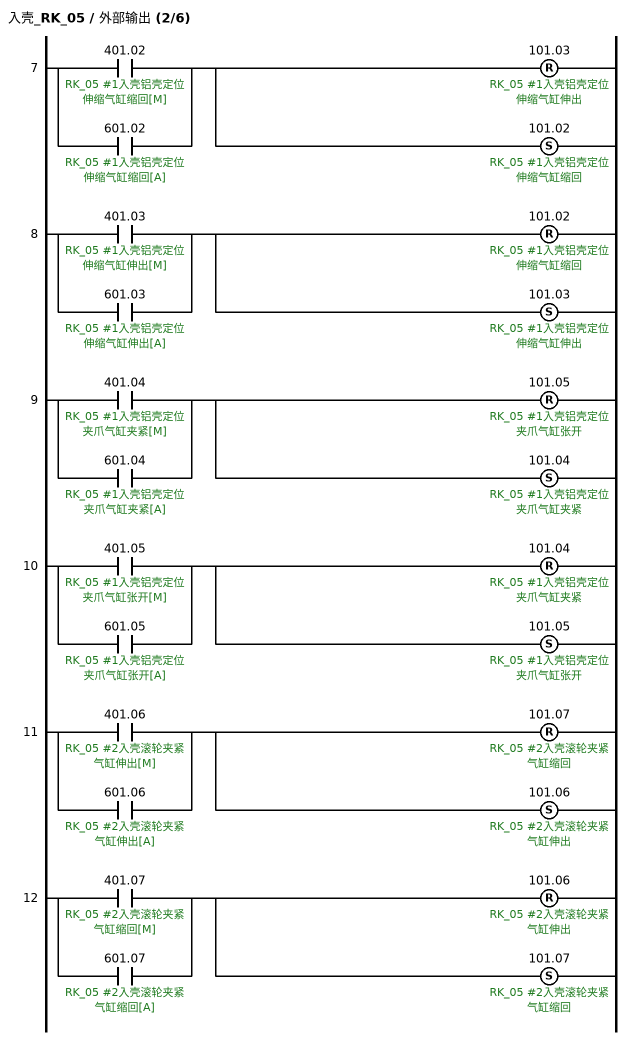
; [picture p504: 入壳_RK_05 / 外部输出, rungs 7-12]
; rung 7
LD 401.02  ; RK_05 #1入壳铝壳定位伸缩气缸缩回[M]
OR 601.02  ; RK_05 #1入壳铝壳定位伸缩气缸缩回[A]
RSET 101.03  ; RK_05 #1入壳铝壳定位伸缩气缸伸出
SET 101.02  ; RK_05 #1入壳铝壳定位伸缩气缸缩回
; rung 8
LD 401.03  ; RK_05 #1入壳铝壳定位伸缩气缸伸出[M]
OR 601.03  ; RK_05 #1入壳铝壳定位伸缩气缸伸出[A]
RSET 101.02  ; RK_05 #1入壳铝壳定位伸缩气缸缩回
SET 101.03  ; RK_05 #1入壳铝壳定位伸缩气缸伸出
; rung 9
LD 401.04  ; RK_05 #1入壳铝壳定位夹爪气缸夹紧[M]
OR 601.04  ; RK_05 #1入壳铝壳定位夹爪气缸夹紧[A]
RSET 101.05  ; RK_05 #1入壳铝壳定位夹爪气缸张开
SET 101.04  ; RK_05 #1入壳铝壳定位夹爪气缸夹紧
; rung 10
LD 401.05  ; RK_05 #1入壳铝壳定位夹爪气缸张开[M]
OR 601.05  ; RK_05 #1入壳铝壳定位夹爪气缸张开[A]
RSET 101.04  ; RK_05 #1入壳铝壳定位夹爪气缸夹紧
SET 101.05  ; RK_05 #1入壳铝壳定位夹爪气缸张开
; rung 11
LD 401.06  ; RK_05 #2入壳滚轮夹紧气缸伸出[M]
OR 601.06  ; RK_05 #2入壳滚轮夹紧气缸伸出[A]
RSET 101.07  ; RK_05 #2入壳滚轮夹紧气缸缩回
SET 101.06  ; RK_05 #2入壳滚轮夹紧气缸伸出
; rung 12
LD 401.07  ; RK_05 #2入壳滚轮夹紧气缸缩回[M]
OR 601.07  ; RK_05 #2入壳滚轮夹紧气缸缩回[A]
RSET 101.06  ; RK_05 #2入壳滚轮夹紧气缸伸出
SET 101.07  ; RK_05 #2入壳滚轮夹紧气缸缩回

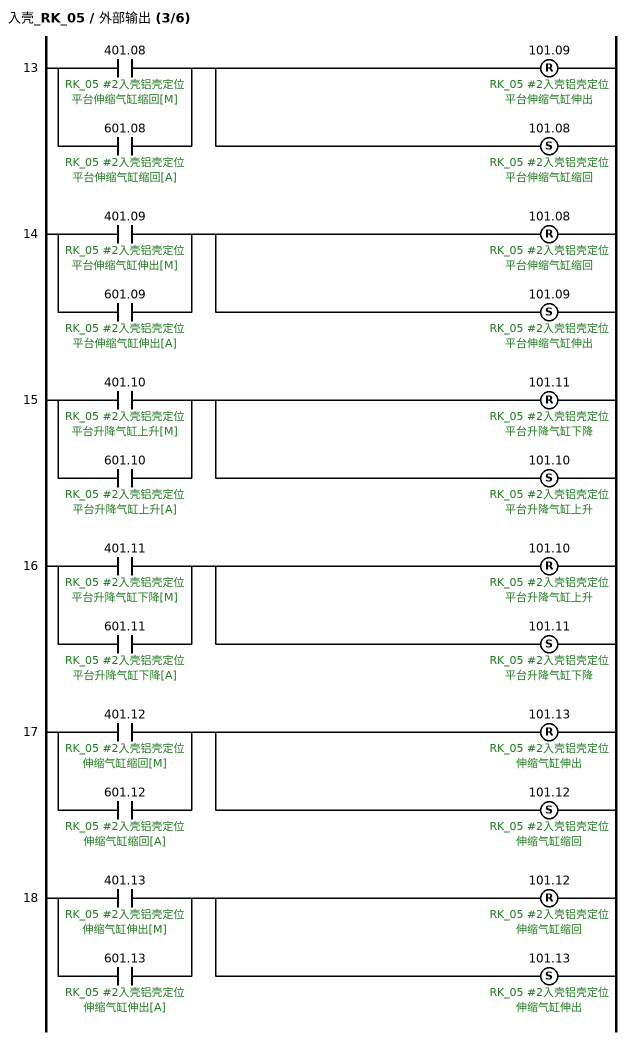
; rung 13
LD 401.08  ; RK_05 #2入壳铝壳定位平台伸缩气缸缩回[M]
OR 601.08  ; RK_05 #2入壳铝壳定位平台伸缩气缸缩回[A]
RSET 101.09  ; RK_05 #2入壳铝壳定位平台伸缩气缸伸出
SET 101.08  ; RK_05 #2入壳铝壳定位平台伸缩气缸缩回
; rung 14
LD 401.09  ; RK_05 #2入壳铝壳定位平台伸缩气缸伸出[M]
OR 601.09  ; RK_05 #2入壳铝壳定位平台伸缩气缸伸出[A]
RSET 101.08  ; RK_05 #2入壳铝壳定位平台伸缩气缸缩回
SET 101.09  ; RK_05 #2入壳铝壳定位平台伸缩气缸伸出
; rung 15
LD 401.10  ; RK_05 #2入壳铝壳定位平台升降气缸上升[M]
OR 601.10  ; RK_05 #2入壳铝壳定位平台升降气缸上升[A]
RSET 101.11  ; RK_05 #2入壳铝壳定位平台升降气缸下降
SET 101.10  ; RK_05 #2入壳铝壳定位平台升降气缸上升
; rung 16
LD 401.11  ; RK_05 #2入壳铝壳定位平台升降气缸下降[M]
OR 601.11  ; RK_05 #2入壳铝壳定位平台升降气缸下降[A]
RSET 101.10  ; RK_05 #2入壳铝壳定位平台升降气缸上升
SET 101.11  ; RK_05 #2入壳铝壳定位平台升降气缸下降
; rung 17
LD 401.12  ; RK_05 #2入壳铝壳定位伸缩气缸缩回[M]
OR 601.12  ; RK_05 #2入壳铝壳定位伸缩气缸缩回[A]
RSET 101.13  ; RK_05 #2入壳铝壳定位伸缩气缸伸出
SET 101.12  ; RK_05 #2入壳铝壳定位伸缩气缸缩回
; rung 18
LD 401.13  ; RK_05 #2入壳铝壳定位伸缩气缸伸出[M]
OR 601.13  ; RK_05 #2入壳铝壳定位伸缩气缸伸出[A]
RSET 101.12  ; RK_05 #2入壳铝壳定位伸缩气缸缩回
SET 101.13  ; RK_05 #2入壳铝壳定位伸缩气缸伸出

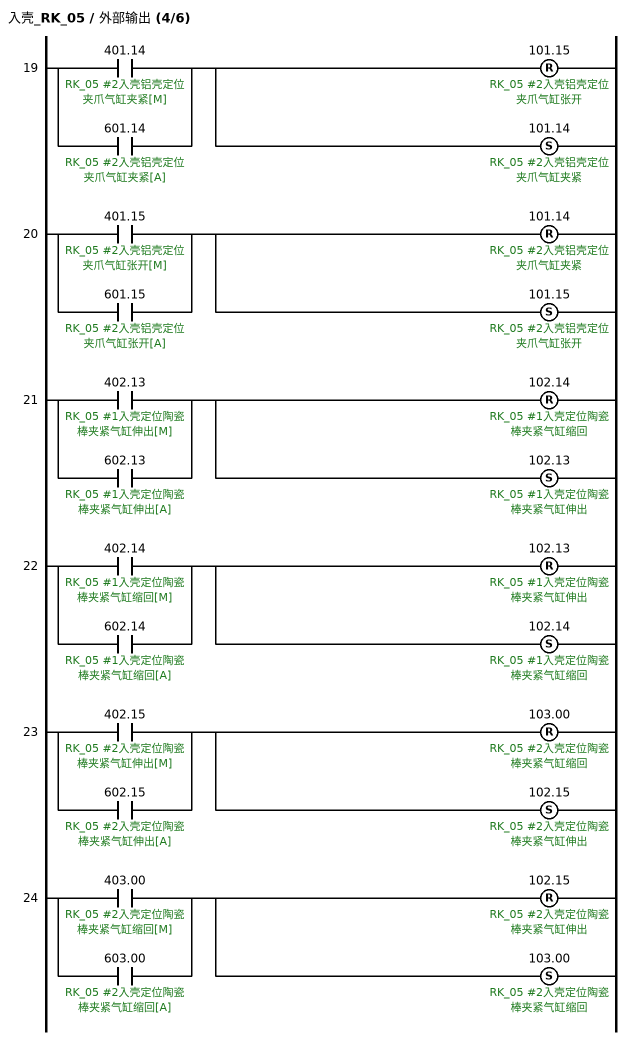
; rung 19
LD 401.14  ; RK_05 #2入壳铝壳定位夹爪气缸夹紧[M]
OR 601.14  ; RK_05 #2入壳铝壳定位夹爪气缸夹紧[A]
RSET 101.15  ; RK_05 #2入壳铝壳定位夹爪气缸张开
SET 101.14  ; RK_05 #2入壳铝壳定位夹爪气缸夹紧
; rung 20
LD 401.15  ; RK_05 #2入壳铝壳定位夹爪气缸张开[M]
OR 601.15  ; RK_05 #2入壳铝壳定位夹爪气缸张开[A]
RSET 101.14  ; RK_05 #2入壳铝壳定位夹爪气缸夹紧
SET 101.15  ; RK_05 #2入壳铝壳定位夹爪气缸张开
; rung 21
LD 402.13  ; RK_05 #1入壳定位陶瓷棒夹紧气缸伸出[M]
OR 602.13  ; RK_05 #1入壳定位陶瓷棒夹紧气缸伸出[A]
RSET 102.14  ; RK_05 #1入壳定位陶瓷棒夹紧气缸缩回
SET 102.13  ; RK_05 #1入壳定位陶瓷棒夹紧气缸伸出
; rung 22
LD 402.14  ; RK_05 #1入壳定位陶瓷棒夹紧气缸缩回[M]
OR 602.14  ; RK_05 #1入壳定位陶瓷棒夹紧气缸缩回[A]
RSET 102.13  ; RK_05 #1入壳定位陶瓷棒夹紧气缸伸出
SET 102.14  ; RK_05 #1入壳定位陶瓷棒夹紧气缸缩回
; rung 23
LD 402.15  ; RK_05 #2入壳定位陶瓷棒夹紧气缸伸出[M]
OR 602.15  ; RK_05 #2入壳定位陶瓷棒夹紧气缸伸出[A]
RSET 103.00  ; RK_05 #2入壳定位陶瓷棒夹紧气缸缩回
SET 102.15  ; RK_05 #2入壳定位陶瓷棒夹紧气缸伸出
; rung 24
LD 403.00  ; RK_05 #2入壳定位陶瓷棒夹紧气缸缩回[M]
OR 603.00  ; RK_05 #2入壳定位陶瓷棒夹紧气缸缩回[A]
RSET 102.15  ; RK_05 #2入壳定位陶瓷棒夹紧气缸伸出
SET 103.00  ; RK_05 #2入壳定位陶瓷棒夹紧气缸缩回

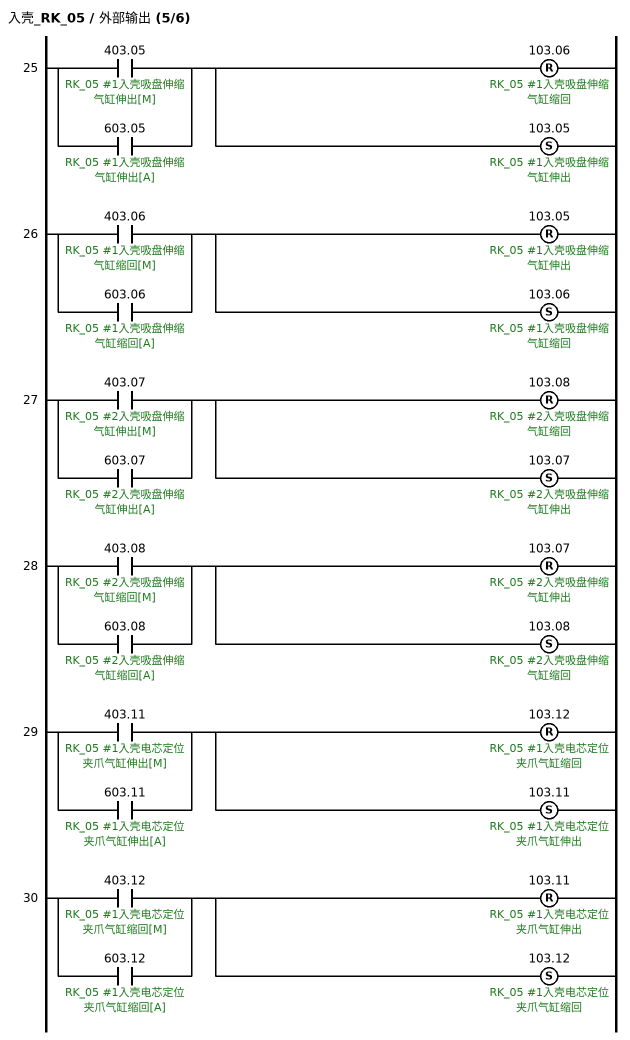
; rung 25
LD 403.05  ; RK_05 #1入壳吸盘伸缩气缸伸出[M]
OR 603.05  ; RK_05 #1入壳吸盘伸缩气缸伸出[A]
RSET 103.06  ; RK_05 #1入壳吸盘伸缩气缸缩回
SET 103.05  ; RK_05 #1入壳吸盘伸缩气缸伸出
; rung 26
LD 403.06  ; RK_05 #1入壳吸盘伸缩气缸缩回[M]
OR 603.06  ; RK_05 #1入壳吸盘伸缩气缸缩回[A]
RSET 103.05  ; RK_05 #1入壳吸盘伸缩气缸伸出
SET 103.06  ; RK_05 #1入壳吸盘伸缩气缸缩回
; rung 27
LD 403.07  ; RK_05 #2入壳吸盘伸缩气缸伸出[M]
OR 603.07  ; RK_05 #2入壳吸盘伸缩气缸伸出[A]
RSET 103.08  ; RK_05 #2入壳吸盘伸缩气缸缩回
SET 103.07  ; RK_05 #2入壳吸盘伸缩气缸伸出
; rung 28
LD 403.08  ; RK_05 #2入壳吸盘伸缩气缸缩回[M]
OR 603.08  ; RK_05 #2入壳吸盘伸缩气缸缩回[A]
RSET 103.07  ; RK_05 #2入壳吸盘伸缩气缸伸出
SET 103.08  ; RK_05 #2入壳吸盘伸缩气缸缩回
; rung 29
LD 403.11  ; RK_05 #1入壳电芯定位夹爪气缸伸出[M]
OR 603.11  ; RK_05 #1入壳电芯定位夹爪气缸伸出[A]
RSET 103.12  ; RK_05 #1入壳电芯定位夹爪气缸缩回
SET 103.11  ; RK_05 #1入壳电芯定位夹爪气缸伸出
; rung 30
LD 403.12  ; RK_05 #1入壳电芯定位夹爪气缸缩回[M]
OR 603.12  ; RK_05 #1入壳电芯定位夹爪气缸缩回[A]
RSET 103.11  ; RK_05 #1入壳电芯定位夹爪气缸伸出
SET 103.12  ; RK_05 #1入壳电芯定位夹爪气缸缩回

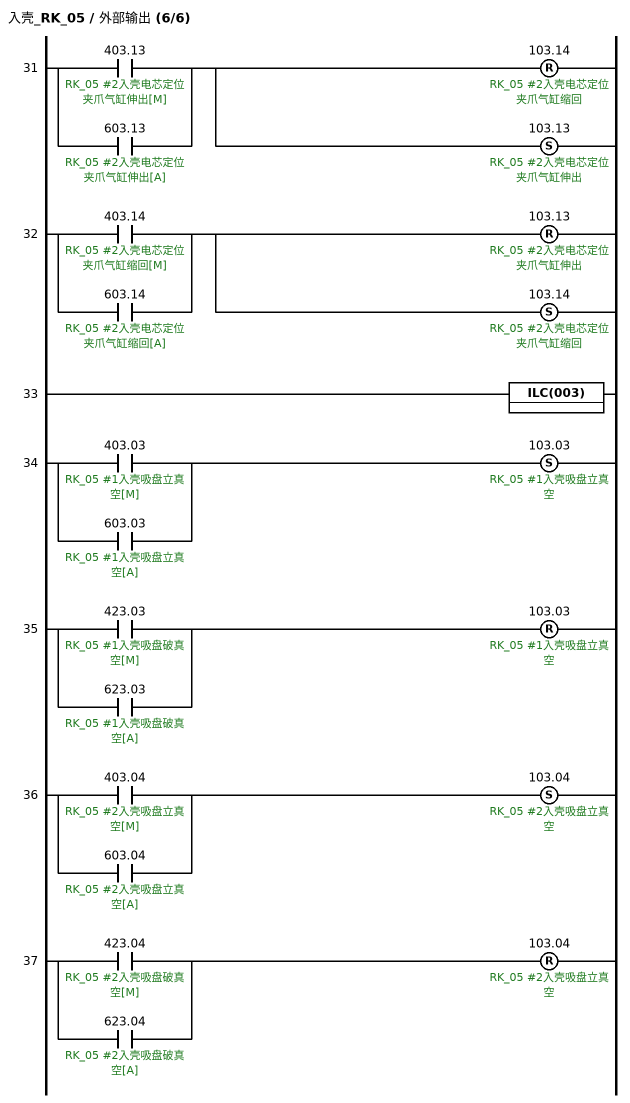
; rung 31
LD 403.13  ; RK_05 #2入壳电芯定位夹爪气缸伸出[M]
OR 603.13  ; RK_05 #2入壳电芯定位夹爪气缸伸出[A]
RSET 103.14  ; RK_05 #2入壳电芯定位夹爪气缸缩回
SET 103.13  ; RK_05 #2入壳电芯定位夹爪气缸伸出
; rung 32
LD 403.14  ; RK_05 #2入壳电芯定位夹爪气缸缩回[M]
OR 603.14  ; RK_05 #2入壳电芯定位夹爪气缸缩回[A]
RSET 103.13  ; RK_05 #2入壳电芯定位夹爪气缸伸出
SET 103.14  ; RK_05 #2入壳电芯定位夹爪气缸缩回
; rung 33
ILC(003)
; rung 34
LD 403.03  ; RK_05 #1入壳吸盘立真空[M]
OR 603.03  ; RK_05 #1入壳吸盘立真空[A]
SET 103.03  ; RK_05 #1入壳吸盘立真空
; rung 35
LD 423.03  ; RK_05 #1入壳吸盘破真空[M]
OR 623.03  ; RK_05 #1入壳吸盘破真空[A]
RSET 103.03  ; RK_05 #1入壳吸盘立真空
; rung 36
LD 403.04  ; RK_05 #2入壳吸盘立真空[M]
OR 603.04  ; RK_05 #2入壳吸盘立真空[A]
SET 103.04  ; RK_05 #2入壳吸盘立真空
; rung 37
LD 423.04  ; RK_05 #2入壳吸盘破真空[M]
OR 623.04  ; RK_05 #2入壳吸盘破真空[A]
RSET 103.04  ; RK_05 #2入壳吸盘立真空

### Section END
; rung 0
END(001)

## Program 电池上下料_RK_06 (cyclic task 6)

### Section Main

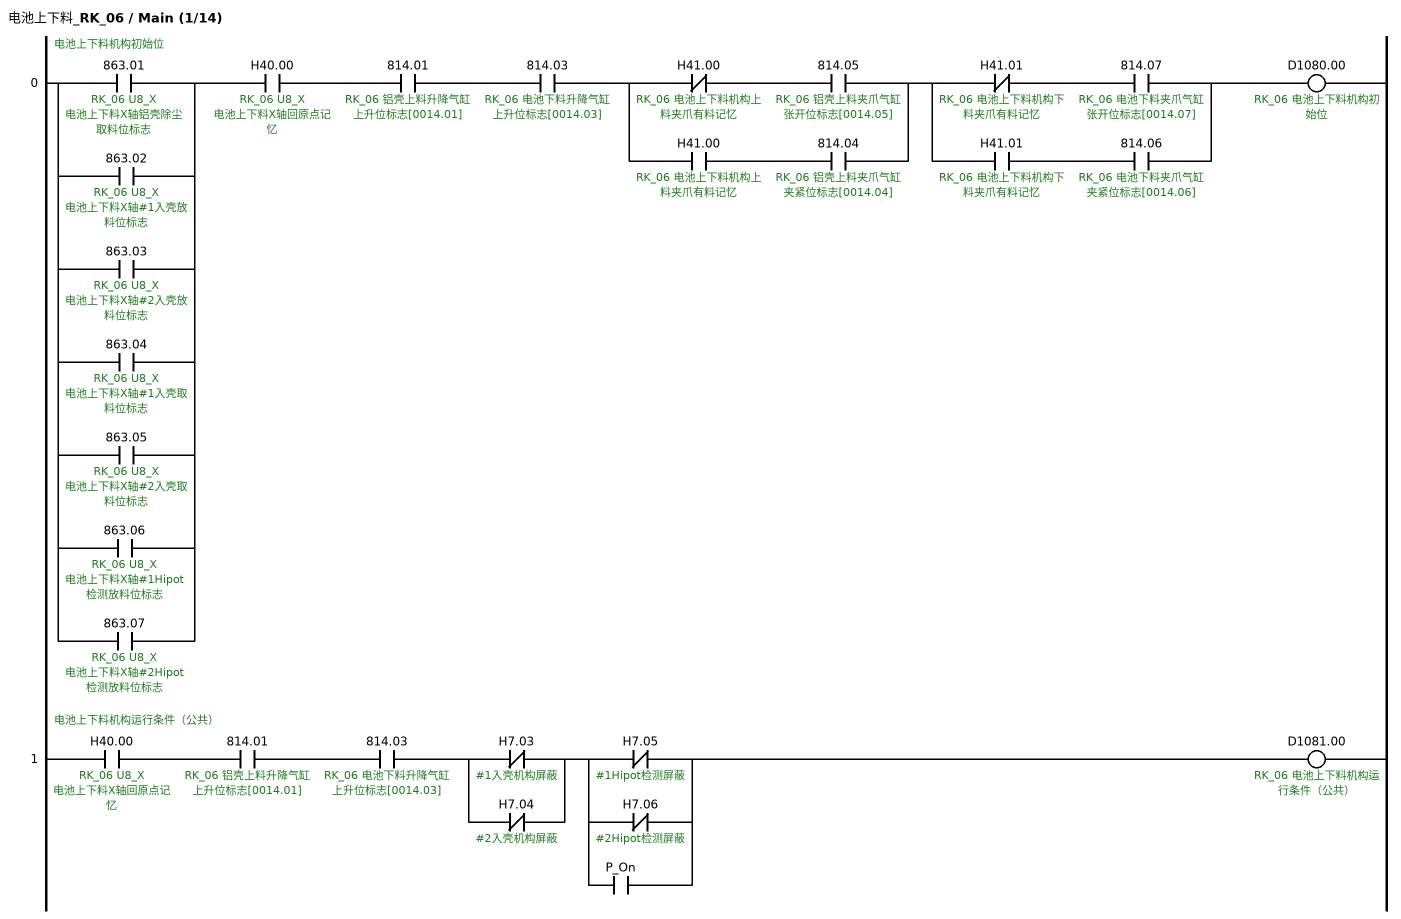
; rung 0: 电池上下料机构初始位
LD 863.01  ; RK_06 U8_X 电池上下料X轴铝壳除尘取料位标志
OR 863.02  ; RK_06 U8_X 电池上下料X轴#1入壳放料位标志
OR 863.03  ; RK_06 U8_X 电池上下料X轴#2入壳放料位标志
OR 863.04  ; RK_06 U8_X 电池上下料X轴#1入壳取料位标志
OR 863.05  ; RK_06 U8_X 电池上下料X轴#2入壳取料位标志
OR 863.06  ; RK_06 U8_X 电池上下料X轴#1Hipot检测放料位标志
OR 863.07  ; RK_06 U8_X 电池上下料X轴#2Hipot检测放料位标志
AND H40.00  ; RK_06 U8_X 电池上下料X轴回原点记忆
AND 814.01  ; RK_06 铝壳上料升降气缸上升位标志[0014.01]
AND 814.03  ; RK_06 电池下料升降气缸上升位标志[0014.03]
LDNOT H41.00  ; RK_06 电池上下料机构上料夹爪有料记忆
AND 814.05  ; RK_06 铝壳上料夹爪气缸张开位标志[0014.05]
LD H41.00  ; RK_06 电池上下料机构上料夹爪有料记忆
AND 814.04  ; RK_06 铝壳上料夹爪气缸夹紧位标志[0014.04]
ORLD
ANDLD
LDNOT H41.01  ; RK_06 电池上下料机构下料夹爪有料记忆
AND 814.07  ; RK_06 电池下料夹爪气缸张开位标志[0014.07]
LD H41.01  ; RK_06 电池上下料机构下料夹爪有料记忆
AND 814.06  ; RK_06 电池下料夹爪气缸夹紧位标志[0014.06]
ORLD
ANDLD
OUT D1080.00  ; RK_06 电池上下料机构初始位
; rung 1: 电池上下料机构运行条件（公共）
LD H40.00  ; RK_06 U8_X 电池上下料X轴回原点记忆
AND 814.01  ; RK_06 铝壳上料升降气缸上升位标志[0014.01]
AND 814.03  ; RK_06 电池下料升降气缸上升位标志[0014.03]
LDNOT H7.03  ; #1入壳机构屏蔽
ORNOT H7.04  ; #2入壳机构屏蔽
ANDLD
LDNOT H7.05  ; #1Hipot检测屏蔽
ORNOT H7.06  ; #2Hipot检测屏蔽
OR P_On
ANDLD
OUT D1081.00  ; RK_06 电池上下料机构运行条件（公共）

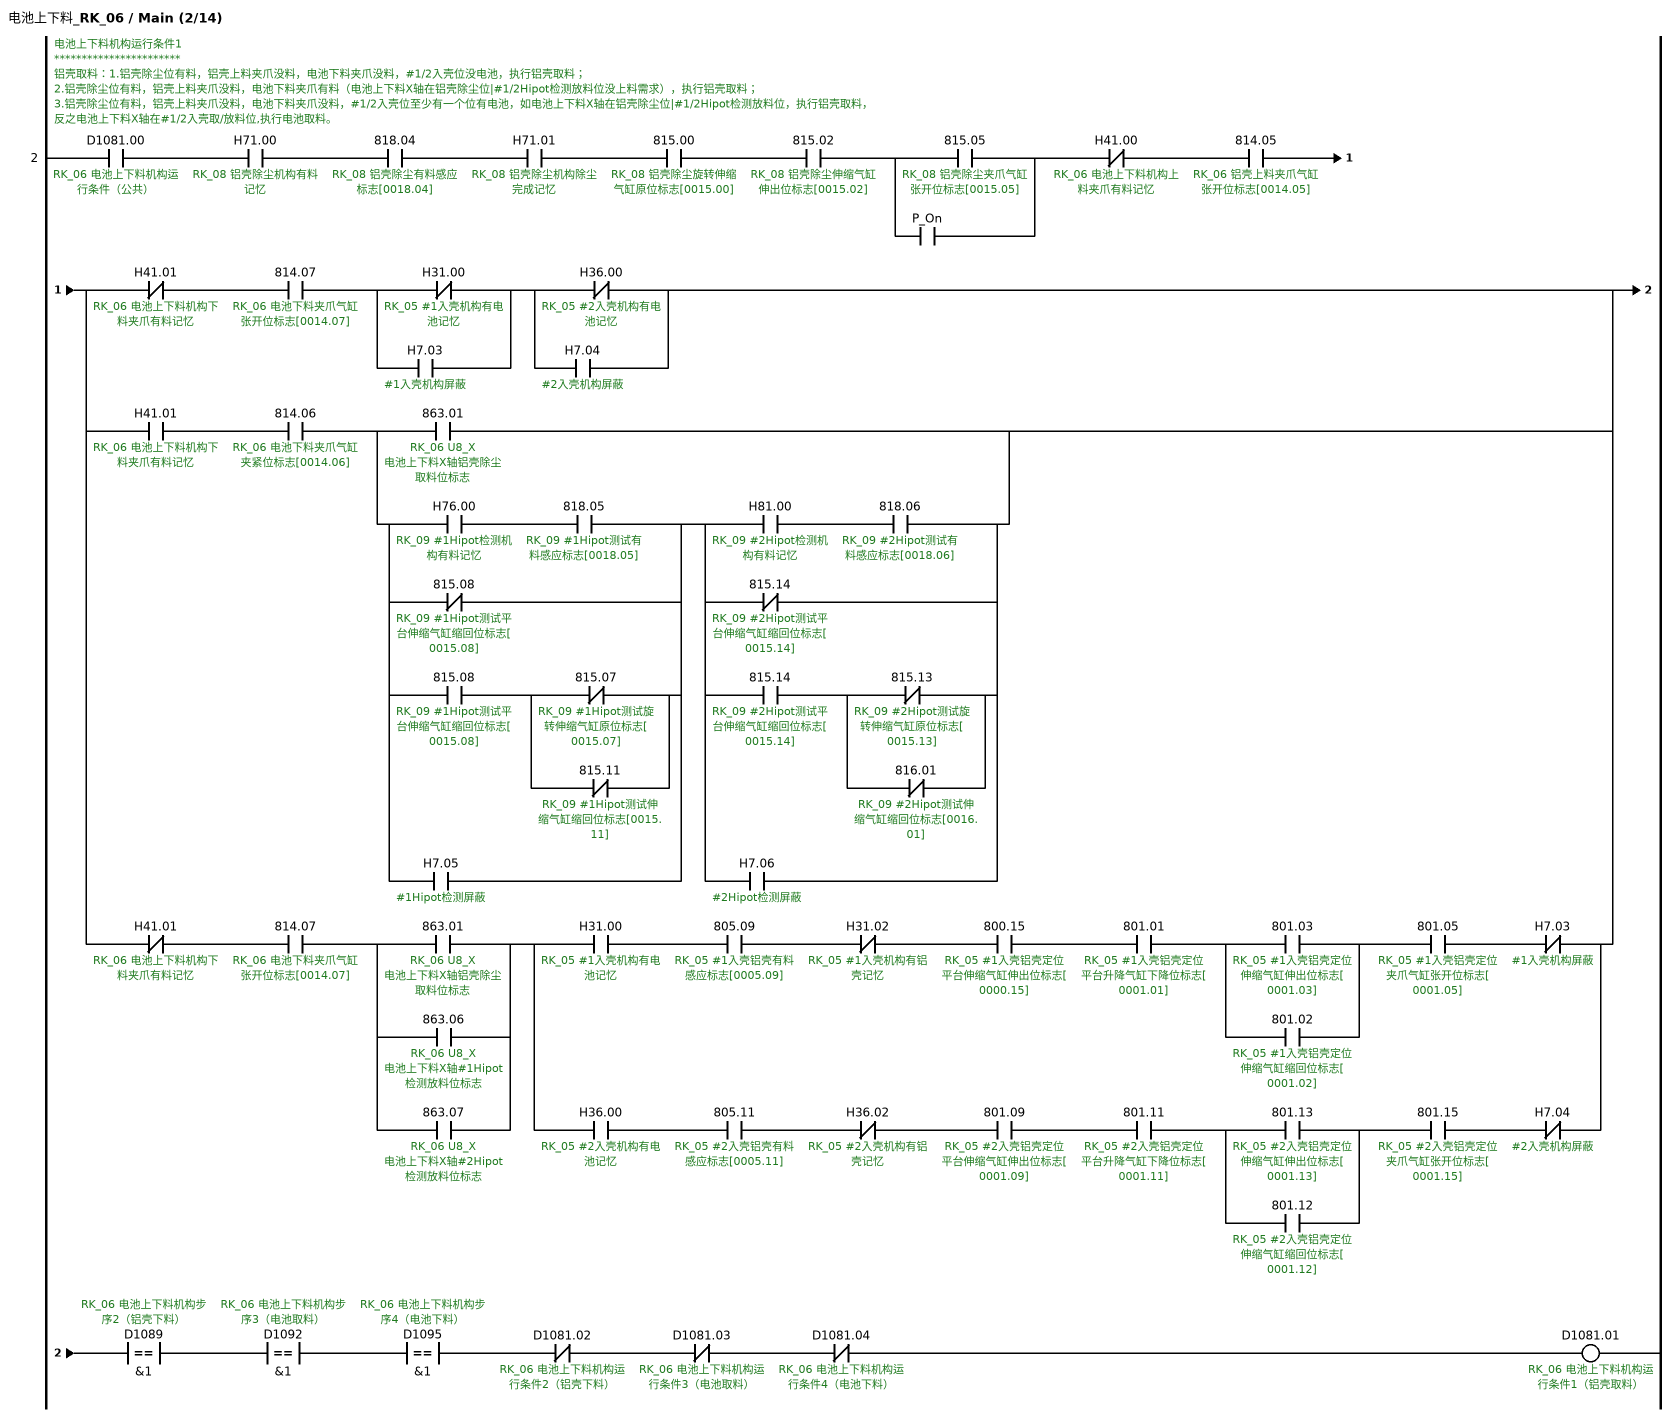
; rung 2: 电池上下料机构运行条件1 / *********************** / 铝壳取料：1.铝壳除尘位有料，铝壳上料夹爪没料，电池下料夹爪没料，#1/2入壳位没电池，执行铝壳取料； / 2.铝壳除尘位有料，铝壳上料夹爪没料，电池下料夹爪有料（电池上下料X轴在铝壳除尘位|#1/2Hipot检测放料位没上料需求），执行铝壳取料； / 3.铝壳除尘位有料，铝壳上料夹爪没料，电池下料夹爪没料，#1/2入壳位至少有一个位有电池，如电池上下料X轴在铝壳除尘位|#1/2Hipot检测放料位，执行铝壳取料， / 反之电池上下料X轴在#1/2入壳取/放料位,执行电池取料。
LD D1081.00  ; RK_06 电池上下料机构运行条件（公共）
AND H71.00  ; RK_08 铝壳除尘机构有料记忆
AND 818.04  ; RK_08 铝壳除尘有料感应标志[0018.04]
AND H71.01  ; RK_08 铝壳除尘机构除尘完成记忆
AND 815.00  ; RK_08 铝壳除尘旋转伸缩气缸原位标志[0015.00]
AND 815.02  ; RK_08 铝壳除尘伸缩气缸伸出位标志[0015.02]
LD 815.05  ; RK_08 铝壳除尘夹爪气缸张开位标志[0015.05]
OR P_On
ANDLD
ANDNOT H41.00  ; RK_06 电池上下料机构上料夹爪有料记忆
AND 814.05  ; RK_06 铝壳上料夹爪气缸张开位标志[0014.05]
LDNOT H41.01  ; RK_06 电池上下料机构下料夹爪有料记忆
AND 814.07  ; RK_06 电池下料夹爪气缸张开位标志[0014.07]
LDNOT H31.00  ; RK_05 #1入壳机构有电池记忆
OR H7.03  ; #1入壳机构屏蔽
ANDLD
LDNOT H36.00  ; RK_05 #2入壳机构有电池记忆
OR H7.04  ; #2入壳机构屏蔽
ANDLD
LD H41.01  ; RK_06 电池上下料机构下料夹爪有料记忆
AND 814.06  ; RK_06 电池下料夹爪气缸夹紧位标志[0014.06]
LD 863.01  ; RK_06 U8_X 电池上下料X轴铝壳除尘取料位标志
LD H76.00  ; RK_09 #1Hipot检测机构有料记忆
AND 818.05  ; RK_09 #1Hipot测试有料感应标志[0018.05]
ORNOT 815.08  ; RK_09 #1Hipot测试平台伸缩气缸缩回位标志[0015.08]
LD 815.08  ; RK_09 #1Hipot测试平台伸缩气缸缩回位标志[0015.08]
LDNOT 815.07  ; RK_09 #1Hipot测试旋转伸缩气缸原位标志[0015.07]
ORNOT 815.11  ; RK_09 #1Hipot测试伸缩气缸缩回位标志[0015.11]
ANDLD
ORLD
OR H7.05  ; #1Hipot检测屏蔽
LD H81.00  ; RK_09 #2Hipot检测机构有料记忆
AND 818.06  ; RK_09 #2Hipot测试有料感应标志[0018.06]
ORNOT 815.14  ; RK_09 #2Hipot测试平台伸缩气缸缩回位标志[0015.14]
LD 815.14  ; RK_09 #2Hipot测试平台伸缩气缸缩回位标志[0015.14]
LDNOT 815.13  ; RK_09 #2Hipot测试旋转伸缩气缸原位标志[0015.13]
ORNOT 816.01  ; RK_09 #2Hipot测试伸缩气缸缩回位标志[0016.01]
ANDLD
ORLD
OR H7.06  ; #2Hipot检测屏蔽
ANDLD
ORLD
ANDLD
ORLD
LDNOT H41.01  ; RK_06 电池上下料机构下料夹爪有料记忆
AND 814.07  ; RK_06 电池下料夹爪气缸张开位标志[0014.07]
LD 863.01  ; RK_06 U8_X 电池上下料X轴铝壳除尘取料位标志
OR 863.06  ; RK_06 U8_X 电池上下料X轴#1Hipot检测放料位标志
OR 863.07  ; RK_06 U8_X 电池上下料X轴#2Hipot检测放料位标志
ANDLD
LD H31.00  ; RK_05 #1入壳机构有电池记忆
AND 805.09  ; RK_05 #1入壳铝壳有料感应标志[0005.09]
ANDNOT H31.02  ; RK_05 #1入壳机构有铝壳记忆
AND 800.15  ; RK_05 #1入壳铝壳定位平台伸缩气缸伸出位标志[0000.15]
AND 801.01  ; RK_05 #1入壳铝壳定位平台升降气缸下降位标志[0001.01]
LD 801.03  ; RK_05 #1入壳铝壳定位伸缩气缸伸出位标志[0001.03]
OR 801.02  ; RK_05 #1入壳铝壳定位伸缩气缸缩回位标志[0001.02]
ANDLD
AND 801.05  ; RK_05 #1入壳铝壳定位夹爪气缸张开位标志[0001.05]
ANDNOT H7.03  ; #1入壳机构屏蔽
LD H36.00  ; RK_05 #2入壳机构有电池记忆
AND 805.11  ; RK_05 #2入壳铝壳有料感应标志[0005.11]
ANDNOT H36.02  ; RK_05 #2入壳机构有铝壳记忆
AND 801.09  ; RK_05 #2入壳铝壳定位平台伸缩气缸伸出位标志[0001.09]
AND 801.11  ; RK_05 #2入壳铝壳定位平台升降气缸下降位标志[0001.11]
LD 801.13  ; RK_05 #2入壳铝壳定位伸缩气缸伸出位标志[0001.13]
OR 801.12  ; RK_05 #2入壳铝壳定位伸缩气缸缩回位标志[0001.12]
ANDLD
AND 801.15  ; RK_05 #2入壳铝壳定位夹爪气缸张开位标志[0001.15]
ANDNOT H7.04  ; #2入壳机构屏蔽
ORLD
ANDLD
ORLD
ANDLD
AND=(300) D1089 &1  ; RK_06 电池上下料机构步序2（铝壳下料）
AND=(300) D1092 &1  ; RK_06 电池上下料机构步序3（电池取料）
AND=(300) D1095 &1  ; RK_06 电池上下料机构步序4（电池下料）
ANDNOT D1081.02  ; RK_06 电池上下料机构运行条件2（铝壳下料）
ANDNOT D1081.03  ; RK_06 电池上下料机构运行条件3（电池取料）
ANDNOT D1081.04  ; RK_06 电池上下料机构运行条件4（电池下料）
OUT D1081.01  ; RK_06 电池上下料机构运行条件1（铝壳取料）

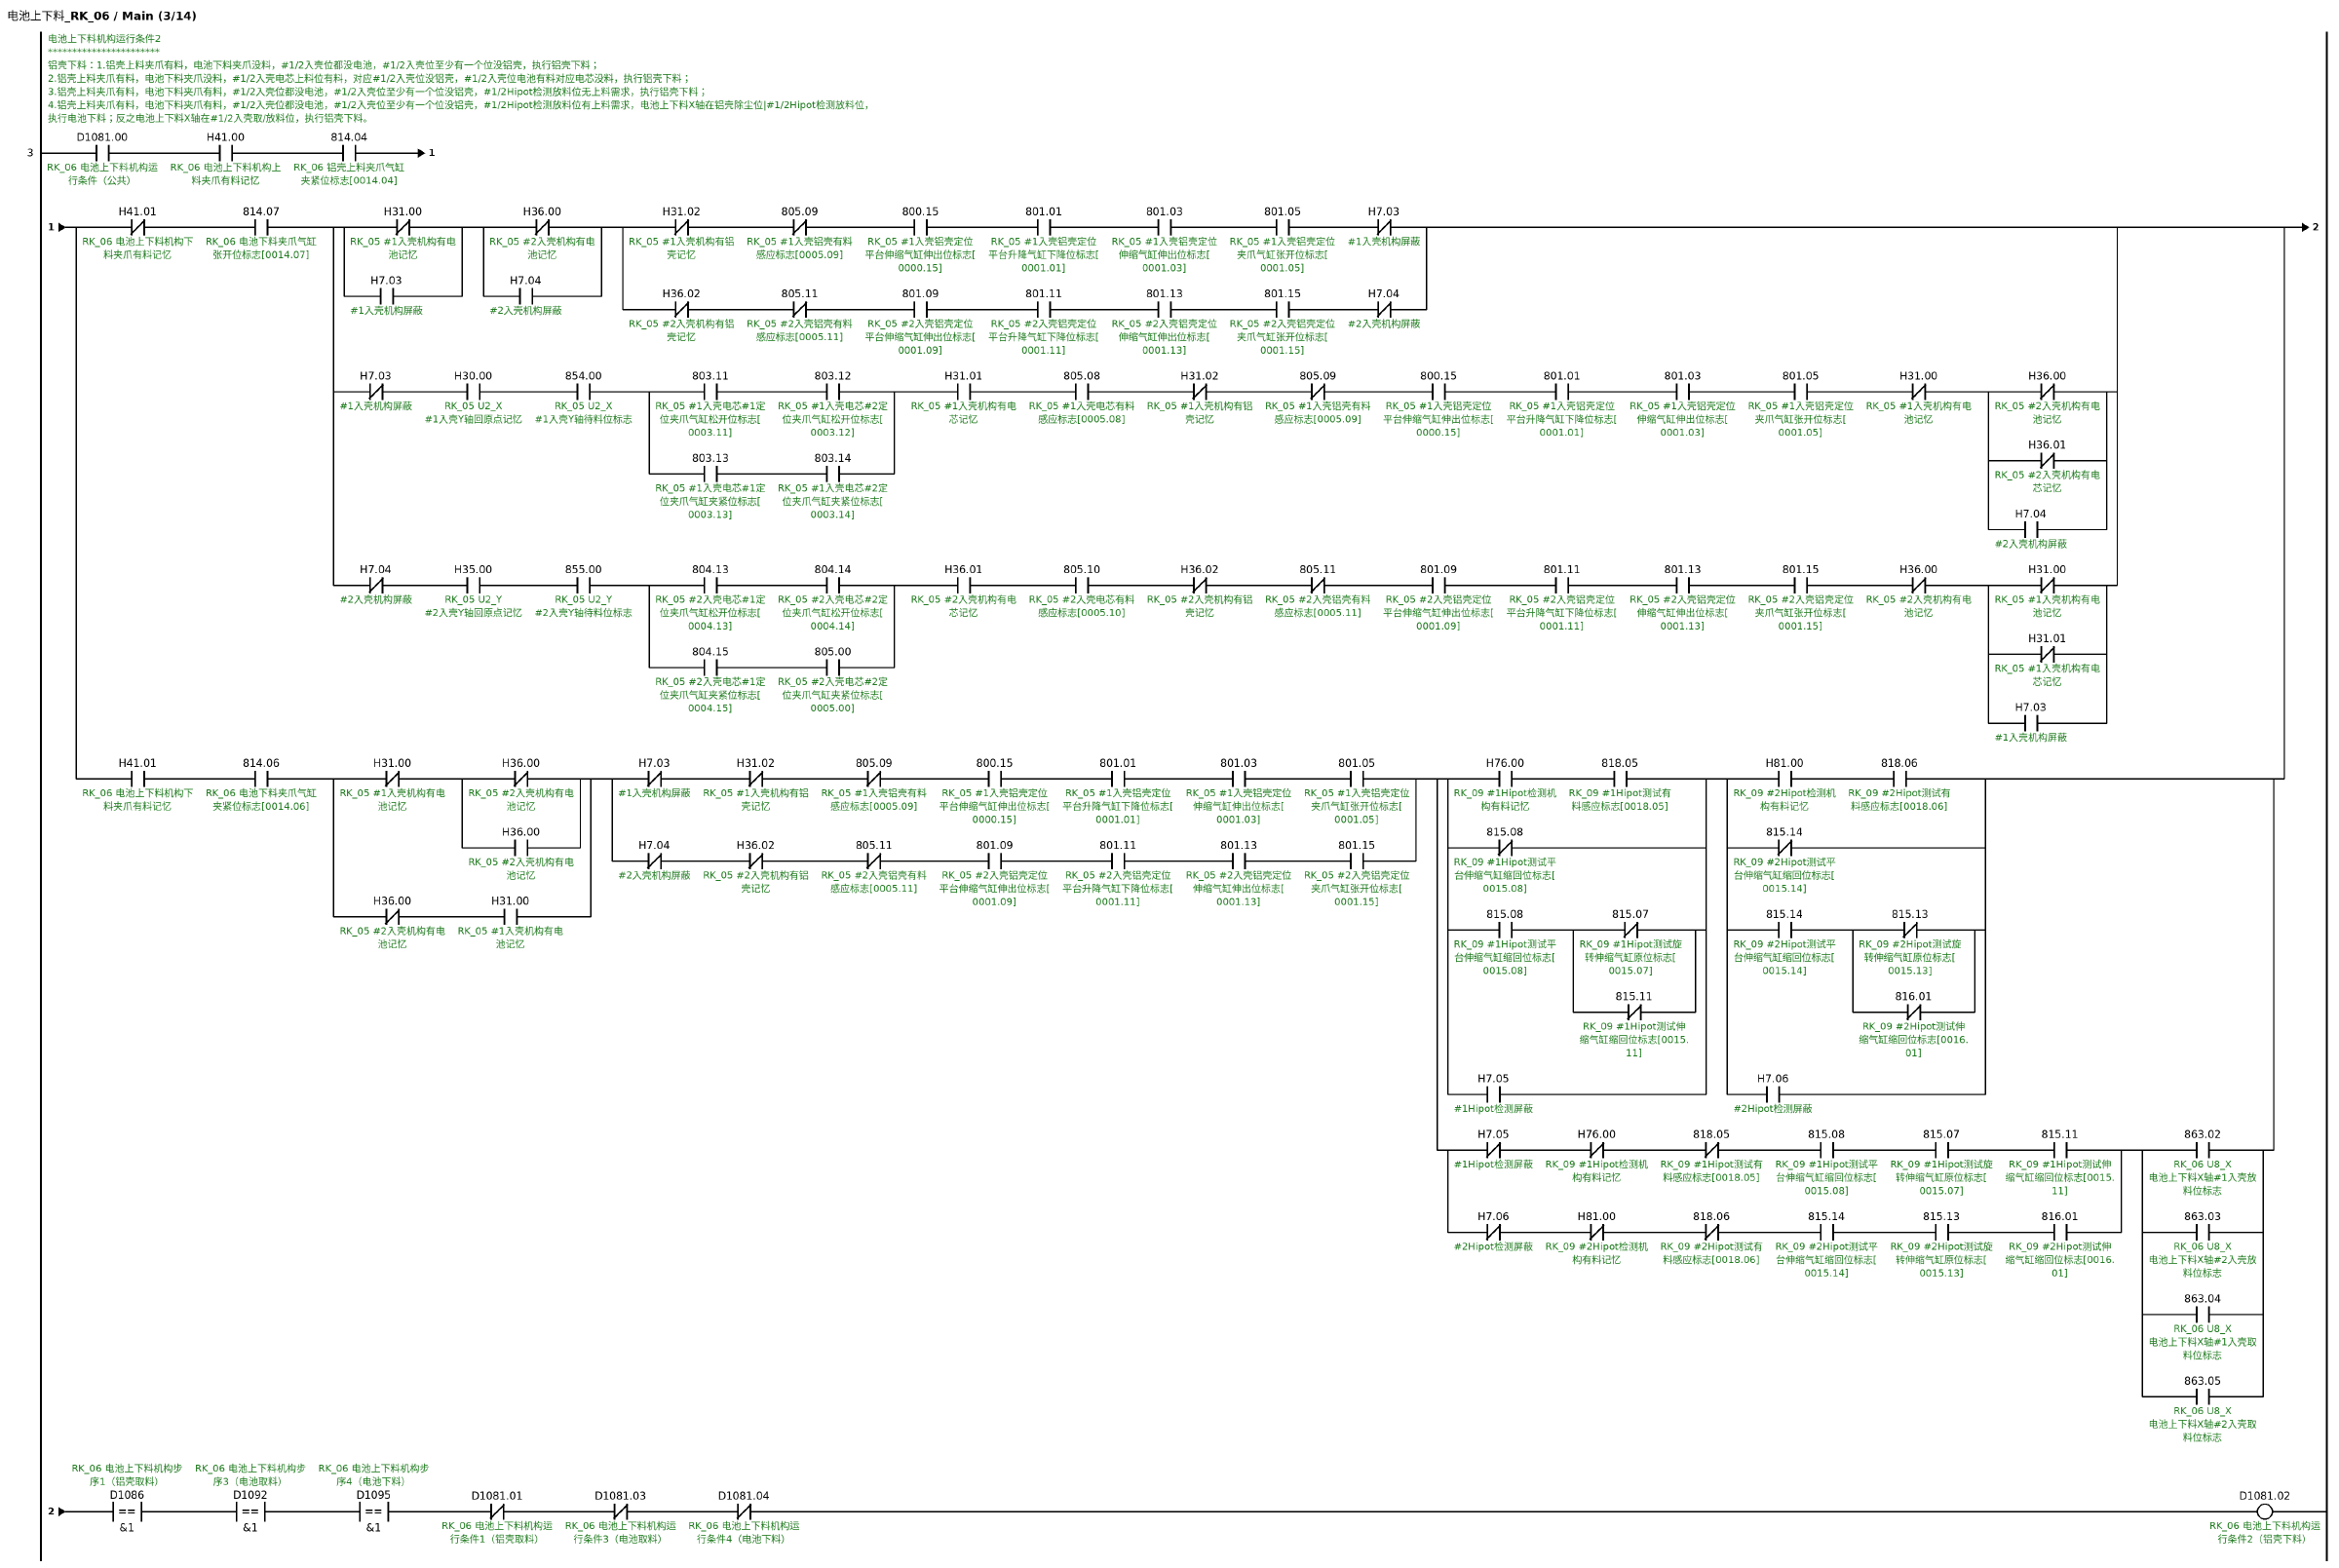
; rung 3: 电池上下料机构运行条件2 / *********************** / 铝壳下料：1.铝壳上料夹爪有料，电池下料夹爪没料，#1/2入壳位都没电池，#1/2入壳位至少有一个位没铝壳，执行铝壳下料； / 2.铝壳上料夹爪有料，电池下料夹爪没料，#1/2入壳电芯上料位有料，对应#1/2入壳位没铝壳，#1/2入壳位电池有料对应电芯没料，执行铝壳下料； / 3.铝壳上料夹爪有料，电池下料夹爪有料，#1/2入壳位都没电池，#1/2入壳位至少有一个位没铝壳，#1/2Hipot检测放料位无上料需求，执行铝壳下料； / 4.铝壳上料夹爪有料，电池下料夹爪有料，#1/2入壳位都没电池，#1/2入壳位至少有一个位没铝壳，#1/2Hipot检测放料位有上料需求，电池上下料X轴在铝壳除尘位|#1/2Hipot检测放料位， / 执行电池下料；反之电池上下料X轴在#1/2入壳取/放料位，执行铝壳下料。
LD D1081.00  ; RK_06 电池上下料机构运行条件（公共）
AND H41.00  ; RK_06 电池上下料机构上料夹爪有料记忆
AND 814.04  ; RK_06 铝壳上料夹爪气缸夹紧位标志[0014.04]
LDNOT H41.01  ; RK_06 电池上下料机构下料夹爪有料记忆
AND 814.07  ; RK_06 电池下料夹爪气缸张开位标志[0014.07]
LDNOT H31.00  ; RK_05 #1入壳机构有电池记忆
OR H7.03  ; #1入壳机构屏蔽
LDNOT H36.00  ; RK_05 #2入壳机构有电池记忆
OR H7.04  ; #2入壳机构屏蔽
ANDLD
LDNOT H31.02  ; RK_05 #1入壳机构有铝壳记忆
ANDNOT 805.09  ; RK_05 #1入壳铝壳有料感应标志[0005.09]
AND 800.15  ; RK_05 #1入壳铝壳定位平台伸缩气缸伸出位标志[0000.15]
AND 801.01  ; RK_05 #1入壳铝壳定位平台升降气缸下降位标志[0001.01]
AND 801.03  ; RK_05 #1入壳铝壳定位伸缩气缸伸出位标志[0001.03]
AND 801.05  ; RK_05 #1入壳铝壳定位夹爪气缸张开位标志[0001.05]
ANDNOT H7.03  ; #1入壳机构屏蔽
LDNOT H36.02  ; RK_05 #2入壳机构有铝壳记忆
ANDNOT 805.11  ; RK_05 #2入壳铝壳有料感应标志[0005.11]
AND 801.09  ; RK_05 #2入壳铝壳定位平台伸缩气缸伸出位标志[0001.09]
AND 801.11  ; RK_05 #2入壳铝壳定位平台升降气缸下降位标志[0001.11]
AND 801.13  ; RK_05 #2入壳铝壳定位伸缩气缸伸出位标志[0001.13]
AND 801.15  ; RK_05 #2入壳铝壳定位夹爪气缸张开位标志[0001.15]
ANDNOT H7.04  ; #2入壳机构屏蔽
ORLD
ANDLD
LDNOT H7.03  ; #1入壳机构屏蔽
AND H30.00  ; RK_05 U2_X #1入壳Y轴回原点记忆
AND 854.00  ; RK_05 U2_X #1入壳Y轴待料位标志
LD 803.11  ; RK_05 #1入壳电芯#1定位夹爪气缸松开位标志[0003.11]
AND 803.12  ; RK_05 #1入壳电芯#2定位夹爪气缸松开位标志[0003.12]
LD 803.13  ; RK_05 #1入壳电芯#1定位夹爪气缸夹紧位标志[0003.13]
AND 803.14  ; RK_05 #1入壳电芯#2定位夹爪气缸夹紧位标志[0003.14]
ORLD
ANDLD
AND H31.01  ; RK_05 #1入壳机构有电芯记忆
AND 805.08  ; RK_05 #1入壳电芯有料感应标志[0005.08]
ANDNOT H31.02  ; RK_05 #1入壳机构有铝壳记忆
ANDNOT 805.09  ; RK_05 #1入壳铝壳有料感应标志[0005.09]
AND 800.15  ; RK_05 #1入壳铝壳定位平台伸缩气缸伸出位标志[0000.15]
AND 801.01  ; RK_05 #1入壳铝壳定位平台升降气缸下降位标志[0001.01]
AND 801.03  ; RK_05 #1入壳铝壳定位伸缩气缸伸出位标志[0001.03]
AND 801.05  ; RK_05 #1入壳铝壳定位夹爪气缸张开位标志[0001.05]
ANDNOT H31.00  ; RK_05 #1入壳机构有电池记忆
LDNOT H36.00  ; RK_05 #2入壳机构有电池记忆
ORNOT H36.01  ; RK_05 #2入壳机构有电芯记忆
OR H7.04  ; #2入壳机构屏蔽
ANDLD
ORLD
LDNOT H7.04  ; #2入壳机构屏蔽
AND H35.00  ; RK_05 U2_Y #2入壳Y轴回原点记忆
AND 855.00  ; RK_05 U2_Y #2入壳Y轴待料位标志
LD 804.13  ; RK_05 #2入壳电芯#1定位夹爪气缸松开位标志[0004.13]
AND 804.14  ; RK_05 #2入壳电芯#2定位夹爪气缸松开位标志[0004.14]
LD 804.15  ; RK_05 #2入壳电芯#1定位夹爪气缸夹紧位标志[0004.15]
AND 805.00  ; RK_05 #2入壳电芯#2定位夹爪气缸夹紧位标志[0005.00]
ORLD
ANDLD
AND H36.01  ; RK_05 #2入壳机构有电芯记忆
AND 805.10  ; RK_05 #2入壳电芯有料感应标志[0005.10]
ANDNOT H36.02  ; RK_05 #2入壳机构有铝壳记忆
ANDNOT 805.11  ; RK_05 #2入壳铝壳有料感应标志[0005.11]
AND 801.09  ; RK_05 #2入壳铝壳定位平台伸缩气缸伸出位标志[0001.09]
AND 801.11  ; RK_05 #2入壳铝壳定位平台升降气缸下降位标志[0001.11]
AND 801.13  ; RK_05 #2入壳铝壳定位伸缩气缸伸出位标志[0001.13]
AND 801.15  ; RK_05 #2入壳铝壳定位夹爪气缸张开位标志[0001.15]
ANDNOT H36.00  ; RK_05 #2入壳机构有电池记忆
LDNOT H31.00  ; RK_05 #1入壳机构有电池记忆
ORNOT H31.01  ; RK_05 #1入壳机构有电芯记忆
OR H7.03  ; #1入壳机构屏蔽
ANDLD
ORLD
ANDLD
LD H41.01  ; RK_06 电池上下料机构下料夹爪有料记忆
AND 814.06  ; RK_06 电池下料夹爪气缸夹紧位标志[0014.06]
LDNOT H31.00  ; RK_05 #1入壳机构有电池记忆
LDNOT H36.00  ; RK_05 #2入壳机构有电池记忆
OR H36.00  ; RK_05 #2入壳机构有电池记忆
ANDLD
LDNOT H36.00  ; RK_05 #2入壳机构有电池记忆
AND H31.00  ; RK_05 #1入壳机构有电池记忆
ORLD
ANDLD
LDNOT H7.03  ; #1入壳机构屏蔽
ANDNOT H31.02  ; RK_05 #1入壳机构有铝壳记忆
ANDNOT 805.09  ; RK_05 #1入壳铝壳有料感应标志[0005.09]
AND 800.15  ; RK_05 #1入壳铝壳定位平台伸缩气缸伸出位标志[0000.15]
AND 801.01  ; RK_05 #1入壳铝壳定位平台升降气缸下降位标志[0001.01]
AND 801.03  ; RK_05 #1入壳铝壳定位伸缩气缸伸出位标志[0001.03]
AND 801.05  ; RK_05 #1入壳铝壳定位夹爪气缸张开位标志[0001.05]
LDNOT H7.04  ; #2入壳机构屏蔽
ANDNOT H36.02  ; RK_05 #2入壳机构有铝壳记忆
ANDNOT 805.11  ; RK_05 #2入壳铝壳有料感应标志[0005.11]
AND 801.09  ; RK_05 #2入壳铝壳定位平台伸缩气缸伸出位标志[0001.09]
AND 801.11  ; RK_05 #2入壳铝壳定位平台升降气缸下降位标志[0001.11]
AND 801.13  ; RK_05 #2入壳铝壳定位伸缩气缸伸出位标志[0001.13]
AND 801.15  ; RK_05 #2入壳铝壳定位夹爪气缸张开位标志[0001.15]
ORLD
ANDLD
LD H76.00  ; RK_09 #1Hipot检测机构有料记忆
AND 818.05  ; RK_09 #1Hipot测试有料感应标志[0018.05]
ORNOT 815.08  ; RK_09 #1Hipot测试平台伸缩气缸缩回位标志[0015.08]
LD 815.08  ; RK_09 #1Hipot测试平台伸缩气缸缩回位标志[0015.08]
LDNOT 815.07  ; RK_09 #1Hipot测试旋转伸缩气缸原位标志[0015.07]
ORNOT 815.11  ; RK_09 #1Hipot测试伸缩气缸缩回位标志[0015.11]
ANDLD
ORLD
OR H7.05  ; #1Hipot检测屏蔽
LD H81.00  ; RK_09 #2Hipot检测机构有料记忆
AND 818.06  ; RK_09 #2Hipot测试有料感应标志[0018.06]
ORNOT 815.14  ; RK_09 #2Hipot测试平台伸缩气缸缩回位标志[0015.14]
LD 815.14  ; RK_09 #2Hipot测试平台伸缩气缸缩回位标志[0015.14]
LDNOT 815.13  ; RK_09 #2Hipot测试旋转伸缩气缸原位标志[0015.13]
ORNOT 816.01  ; RK_09 #2Hipot测试伸缩气缸缩回位标志[0016.01]
ANDLD
ORLD
OR H7.06  ; #2Hipot检测屏蔽
ANDLD
LDNOT H7.05  ; #1Hipot检测屏蔽
ANDNOT H76.00  ; RK_09 #1Hipot检测机构有料记忆
ANDNOT 818.05  ; RK_09 #1Hipot测试有料感应标志[0018.05]
AND 815.08  ; RK_09 #1Hipot测试平台伸缩气缸缩回位标志[0015.08]
AND 815.07  ; RK_09 #1Hipot测试旋转伸缩气缸原位标志[0015.07]
AND 815.11  ; RK_09 #1Hipot测试伸缩气缸缩回位标志[0015.11]
LDNOT H7.06  ; #2Hipot检测屏蔽
ANDNOT H81.00  ; RK_09 #2Hipot检测机构有料记忆
ANDNOT 818.06  ; RK_09 #2Hipot测试有料感应标志[0018.06]
AND 815.14  ; RK_09 #2Hipot测试平台伸缩气缸缩回位标志[0015.14]
AND 815.13  ; RK_09 #2Hipot测试旋转伸缩气缸原位标志[0015.13]
AND 816.01  ; RK_09 #2Hipot测试伸缩气缸缩回位标志[0016.01]
ORLD
LD 863.02  ; RK_06 U8_X 电池上下料X轴#1入壳放料位标志
OR 863.03  ; RK_06 U8_X 电池上下料X轴#2入壳放料位标志
OR 863.04  ; RK_06 U8_X 电池上下料X轴#1入壳取料位标志
OR 863.05  ; RK_06 U8_X 电池上下料X轴#2入壳取料位标志
ANDLD
ORLD
ANDLD
ORLD
ANDLD
AND=(300) D1086 &1  ; RK_06 电池上下料机构步序1（铝壳取料）
AND=(300) D1092 &1  ; RK_06 电池上下料机构步序3（电池取料）
AND=(300) D1095 &1  ; RK_06 电池上下料机构步序4（电池下料）
ANDNOT D1081.01  ; RK_06 电池上下料机构运行条件1（铝壳取料）
ANDNOT D1081.03  ; RK_06 电池上下料机构运行条件3（电池取料）
ANDNOT D1081.04  ; RK_06 电池上下料机构运行条件4（电池下料）
OUT D1081.02  ; RK_06 电池上下料机构运行条件2（铝壳下料）

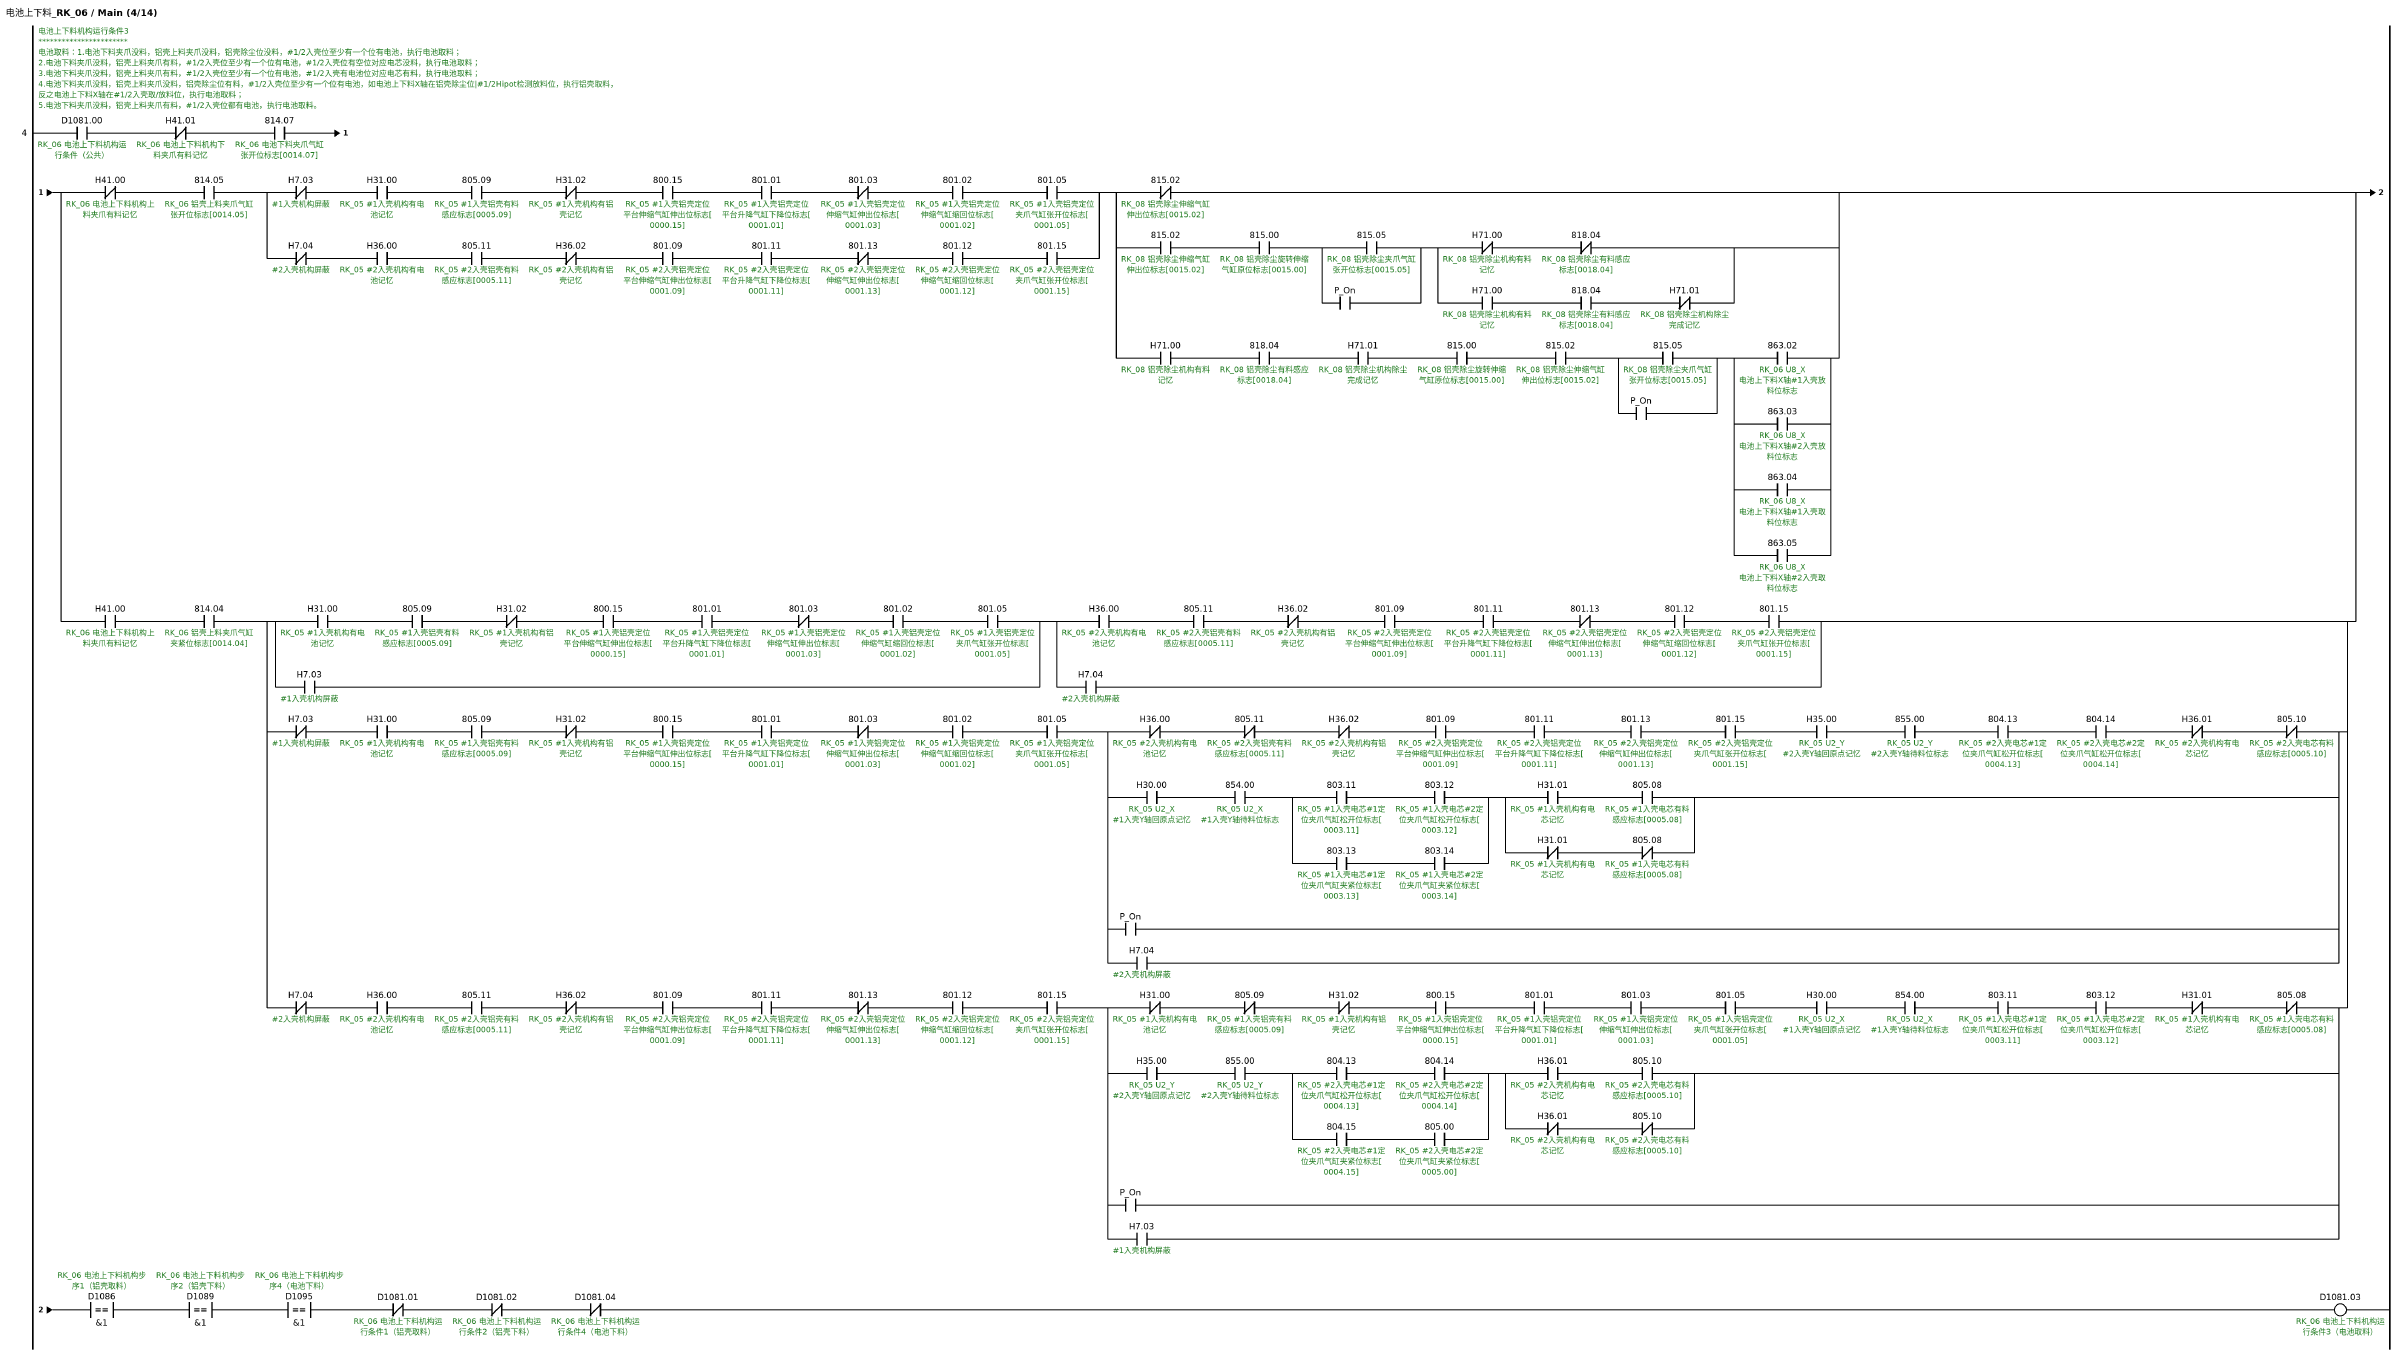
; rung 4: 电池上下料机构运行条件3 / *********************** / 电池取料：1.电池下料夹爪没料，铝壳上料夹爪没料，铝壳除尘位没料，#1/2入壳位至少有一个位有电池，执行电池取料； / 2.电池下料夹爪没料，铝壳上料夹爪有料，#1/2入壳位至少有一个位有电池，#1/2入壳位有空位对应电芯没料，执行电池取料； / 3.电池下料夹爪没料，铝壳上料夹爪有料，#1/2入壳位至少有一个位有电池，#1/2入壳有电池位对应电芯有料，执行电池取料； / 4.电池下料夹爪没料，铝壳上料夹爪没料，铝壳除尘位有料，#1/2入壳位至少有一个位有电池，如电池上下料X轴在铝壳除尘位|#1/2Hipot检测放料位，执行铝壳取料， / 反之电池上下料X轴在#1/2入壳取/放料位，执行电池取料； / 5.电池下料夹爪没料，铝壳上料夹爪有料，#1/2入壳位都有电池，执行电池取料。
LD D1081.00  ; RK_06 电池上下料机构运行条件（公共）
ANDNOT H41.01  ; RK_06 电池上下料机构下料夹爪有料记忆
AND 814.07  ; RK_06 电池下料夹爪气缸张开位标志[0014.07]
LDNOT H41.00  ; RK_06 电池上下料机构上料夹爪有料记忆
AND 814.05  ; RK_06 铝壳上料夹爪气缸张开位标志[0014.05]
LDNOT H7.03  ; #1入壳机构屏蔽
AND H31.00  ; RK_05 #1入壳机构有电池记忆
AND 805.09  ; RK_05 #1入壳铝壳有料感应标志[0005.09]
ANDNOT H31.02  ; RK_05 #1入壳机构有铝壳记忆
AND 800.15  ; RK_05 #1入壳铝壳定位平台伸缩气缸伸出位标志[0000.15]
AND 801.01  ; RK_05 #1入壳铝壳定位平台升降气缸下降位标志[0001.01]
ANDNOT 801.03  ; RK_05 #1入壳铝壳定位伸缩气缸伸出位标志[0001.03]  // 20190306修改（ON改OFF）
AND 801.02  ; RK_05 #1入壳铝壳定位伸缩气缸缩回位标志[0001.02]
AND 801.05  ; RK_05 #1入壳铝壳定位夹爪气缸张开位标志[0001.05]
LDNOT H7.04  ; #2入壳机构屏蔽
AND H36.00  ; RK_05 #2入壳机构有电池记忆
AND 805.11  ; RK_05 #2入壳铝壳有料感应标志[0005.11]
ANDNOT H36.02  ; RK_05 #2入壳机构有铝壳记忆
AND 801.09  ; RK_05 #2入壳铝壳定位平台伸缩气缸伸出位标志[0001.09]
AND 801.11  ; RK_05 #2入壳铝壳定位平台升降气缸下降位标志[0001.11]
ANDNOT 801.13  ; RK_05 #2入壳铝壳定位伸缩气缸伸出位标志[0001.13]  // 20190306修改（ON改OFF）
AND 801.12  ; RK_05 #2入壳铝壳定位伸缩气缸缩回位标志[0001.12]
AND 801.15  ; RK_05 #2入壳铝壳定位夹爪气缸张开位标志[0001.15]
ORLD
ANDLD
LDNOT 815.02  ; RK_08 铝壳除尘伸缩气缸伸出位标志[0015.02]
LD 815.02  ; RK_08 铝壳除尘伸缩气缸伸出位标志[0015.02]
AND 815.00  ; RK_08 铝壳除尘旋转伸缩气缸原位标志[0015.00]
LD 815.05  ; RK_08 铝壳除尘夹爪气缸张开位标志[0015.05]
OR P_On
ANDLD
LDNOT H71.00  ; RK_08 铝壳除尘机构有料记忆
ANDNOT 818.04  ; RK_08 铝壳除尘有料感应标志[0018.04]
LD H71.00  ; RK_08 铝壳除尘机构有料记忆
AND 818.04  ; RK_08 铝壳除尘有料感应标志[0018.04]
ANDNOT H71.01  ; RK_08 铝壳除尘机构除尘完成记忆
ORLD
ANDLD
ORLD
LD H71.00  ; RK_08 铝壳除尘机构有料记忆
AND 818.04  ; RK_08 铝壳除尘有料感应标志[0018.04]
AND H71.01  ; RK_08 铝壳除尘机构除尘完成记忆
AND 815.00  ; RK_08 铝壳除尘旋转伸缩气缸原位标志[0015.00]
AND 815.02  ; RK_08 铝壳除尘伸缩气缸伸出位标志[0015.02]
LD 815.05  ; RK_08 铝壳除尘夹爪气缸张开位标志[0015.05]
OR P_On
ANDLD
LD 863.02  ; RK_06 U8_X 电池上下料X轴#1入壳放料位标志
OR 863.03  ; RK_06 U8_X 电池上下料X轴#2入壳放料位标志
OR 863.04  ; RK_06 U8_X 电池上下料X轴#1入壳取料位标志
OR 863.05  ; RK_06 U8_X 电池上下料X轴#2入壳取料位标志
ANDLD
ORLD
ANDLD
LD H41.00  ; RK_06 电池上下料机构上料夹爪有料记忆
AND 814.04  ; RK_06 铝壳上料夹爪气缸夹紧位标志[0014.04]
LD H31.00  ; RK_05 #1入壳机构有电池记忆
AND 805.09  ; RK_05 #1入壳铝壳有料感应标志[0005.09]
ANDNOT H31.02  ; RK_05 #1入壳机构有铝壳记忆
AND 800.15  ; RK_05 #1入壳铝壳定位平台伸缩气缸伸出位标志[0000.15]
AND 801.01  ; RK_05 #1入壳铝壳定位平台升降气缸下降位标志[0001.01]
ANDNOT 801.03  ; RK_05 #1入壳铝壳定位伸缩气缸伸出位标志[0001.03]
AND 801.02  ; RK_05 #1入壳铝壳定位伸缩气缸缩回位标志[0001.02]
AND 801.05  ; RK_05 #1入壳铝壳定位夹爪气缸张开位标志[0001.05]
OR H7.03  ; #1入壳机构屏蔽
LD H36.00  ; RK_05 #2入壳机构有电池记忆
AND 805.11  ; RK_05 #2入壳铝壳有料感应标志[0005.11]
ANDNOT H36.02  ; RK_05 #2入壳机构有铝壳记忆
AND 801.09  ; RK_05 #2入壳铝壳定位平台伸缩气缸伸出位标志[0001.09]
AND 801.11  ; RK_05 #2入壳铝壳定位平台升降气缸下降位标志[0001.11]
ANDNOT 801.13  ; RK_05 #2入壳铝壳定位伸缩气缸伸出位标志[0001.13]
AND 801.12  ; RK_05 #2入壳铝壳定位伸缩气缸缩回位标志[0001.12]
AND 801.15  ; RK_05 #2入壳铝壳定位夹爪气缸张开位标志[0001.15]
OR H7.04  ; #2入壳机构屏蔽
ANDLD
LDNOT H7.03  ; #1入壳机构屏蔽
AND H31.00  ; RK_05 #1入壳机构有电池记忆
AND 805.09  ; RK_05 #1入壳铝壳有料感应标志[0005.09]
ANDNOT H31.02  ; RK_05 #1入壳机构有铝壳记忆
AND 800.15  ; RK_05 #1入壳铝壳定位平台伸缩气缸伸出位标志[0000.15]
AND 801.01  ; RK_05 #1入壳铝壳定位平台升降气缸下降位标志[0001.01]
ANDNOT 801.03  ; RK_05 #1入壳铝壳定位伸缩气缸伸出位标志[0001.03]
AND 801.02  ; RK_05 #1入壳铝壳定位伸缩气缸缩回位标志[0001.02]
AND 801.05  ; RK_05 #1入壳铝壳定位夹爪气缸张开位标志[0001.05]
LDNOT H36.00  ; RK_05 #2入壳机构有电池记忆
ANDNOT 805.11  ; RK_05 #2入壳铝壳有料感应标志[0005.11]
ANDNOT H36.02  ; RK_05 #2入壳机构有铝壳记忆
AND 801.09  ; RK_05 #2入壳铝壳定位平台伸缩气缸伸出位标志[0001.09]
AND 801.11  ; RK_05 #2入壳铝壳定位平台升降气缸下降位标志[0001.11]
AND 801.13  ; RK_05 #2入壳铝壳定位伸缩气缸伸出位标志[0001.13]
AND 801.15  ; RK_05 #2入壳铝壳定位夹爪气缸张开位标志[0001.15]
AND H35.00  ; RK_05 U2_Y #2入壳Y轴回原点记忆
AND 855.00  ; RK_05 U2_Y #2入壳Y轴待料位标志
AND 804.13  ; RK_05 #2入壳电芯#1定位夹爪气缸松开位标志[0004.13]
AND 804.14  ; RK_05 #2入壳电芯#2定位夹爪气缸松开位标志[0004.14]
ANDNOT H36.01  ; RK_05 #2入壳机构有电芯记忆
ANDNOT 805.10  ; RK_05 #2入壳电芯有料感应标志[0005.10]
LD H30.00  ; RK_05 U2_X #1入壳Y轴回原点记忆
AND 854.00  ; RK_05 U2_X #1入壳Y轴待料位标志
LD 803.11  ; RK_05 #1入壳电芯#1定位夹爪气缸松开位标志[0003.11]
AND 803.12  ; RK_05 #1入壳电芯#2定位夹爪气缸松开位标志[0003.12]
LD 803.13  ; RK_05 #1入壳电芯#1定位夹爪气缸夹紧位标志[0003.13]
AND 803.14  ; RK_05 #1入壳电芯#2定位夹爪气缸夹紧位标志[0003.14]
ORLD
ANDLD
LD H31.01  ; RK_05 #1入壳机构有电芯记忆
AND 805.08  ; RK_05 #1入壳电芯有料感应标志[0005.08]
LDNOT H31.01  ; RK_05 #1入壳机构有电芯记忆
ANDNOT 805.08  ; RK_05 #1入壳电芯有料感应标志[0005.08]
ORLD
ANDLD
ORLD
OR P_On
OR H7.04  ; #2入壳机构屏蔽
ANDLD
ORLD
LDNOT H7.04  ; #2入壳机构屏蔽
AND H36.00  ; RK_05 #2入壳机构有电池记忆
AND 805.11  ; RK_05 #2入壳铝壳有料感应标志[0005.11]
ANDNOT H36.02  ; RK_05 #2入壳机构有铝壳记忆
AND 801.09  ; RK_05 #2入壳铝壳定位平台伸缩气缸伸出位标志[0001.09]
AND 801.11  ; RK_05 #2入壳铝壳定位平台升降气缸下降位标志[0001.11]
ANDNOT 801.13  ; RK_05 #2入壳铝壳定位伸缩气缸伸出位标志[0001.13]
AND 801.12  ; RK_05 #2入壳铝壳定位伸缩气缸缩回位标志[0001.12]
AND 801.15  ; RK_05 #2入壳铝壳定位夹爪气缸张开位标志[0001.15]
LDNOT H31.00  ; RK_05 #1入壳机构有电池记忆
ANDNOT 805.09  ; RK_05 #1入壳铝壳有料感应标志[0005.09]
ANDNOT H31.02  ; RK_05 #1入壳机构有铝壳记忆
AND 800.15  ; RK_05 #1入壳铝壳定位平台伸缩气缸伸出位标志[0000.15]
AND 801.01  ; RK_05 #1入壳铝壳定位平台升降气缸下降位标志[0001.01]
AND 801.03  ; RK_05 #1入壳铝壳定位伸缩气缸伸出位标志[0001.03]
AND 801.05  ; RK_05 #1入壳铝壳定位夹爪气缸张开位标志[0001.05]
AND H30.00  ; RK_05 U2_X #1入壳Y轴回原点记忆
AND 854.00  ; RK_05 U2_X #1入壳Y轴待料位标志
AND 803.11  ; RK_05 #1入壳电芯#1定位夹爪气缸松开位标志[0003.11]
AND 803.12  ; RK_05 #1入壳电芯#2定位夹爪气缸松开位标志[0003.12]
ANDNOT H31.01  ; RK_05 #1入壳机构有电芯记忆
ANDNOT 805.08  ; RK_05 #1入壳电芯有料感应标志[0005.08]
LD H35.00  ; RK_05 U2_Y #2入壳Y轴回原点记忆
AND 855.00  ; RK_05 U2_Y #2入壳Y轴待料位标志
LD 804.13  ; RK_05 #2入壳电芯#1定位夹爪气缸松开位标志[0004.13]
AND 804.14  ; RK_05 #2入壳电芯#2定位夹爪气缸松开位标志[0004.14]
LD 804.15  ; RK_05 #2入壳电芯#1定位夹爪气缸夹紧位标志[0004.15]
AND 805.00  ; RK_05 #2入壳电芯#2定位夹爪气缸夹紧位标志[0005.00]
ORLD
ANDLD
LD H36.01  ; RK_05 #2入壳机构有电芯记忆
AND 805.10  ; RK_05 #2入壳电芯有料感应标志[0005.10]
LDNOT H36.01  ; RK_05 #2入壳机构有电芯记忆
ANDNOT 805.10  ; RK_05 #2入壳电芯有料感应标志[0005.10]
ORLD
ANDLD
ORLD
OR P_On
OR H7.03  ; #1入壳机构屏蔽
ANDLD
ORLD
ANDLD
ORLD
ANDLD
AND=(300) D1086 &1  ; RK_06 电池上下料机构步序1（铝壳取料）
AND=(300) D1089 &1  ; RK_06 电池上下料机构步序2（铝壳下料）
AND=(300) D1095 &1  ; RK_06 电池上下料机构步序4（电池下料）
ANDNOT D1081.01  ; RK_06 电池上下料机构运行条件1（铝壳取料）
ANDNOT D1081.02  ; RK_06 电池上下料机构运行条件2（铝壳下料）
ANDNOT D1081.04  ; RK_06 电池上下料机构运行条件4（电池下料）
OUT D1081.03  ; RK_06 电池上下料机构运行条件3（电池取料）

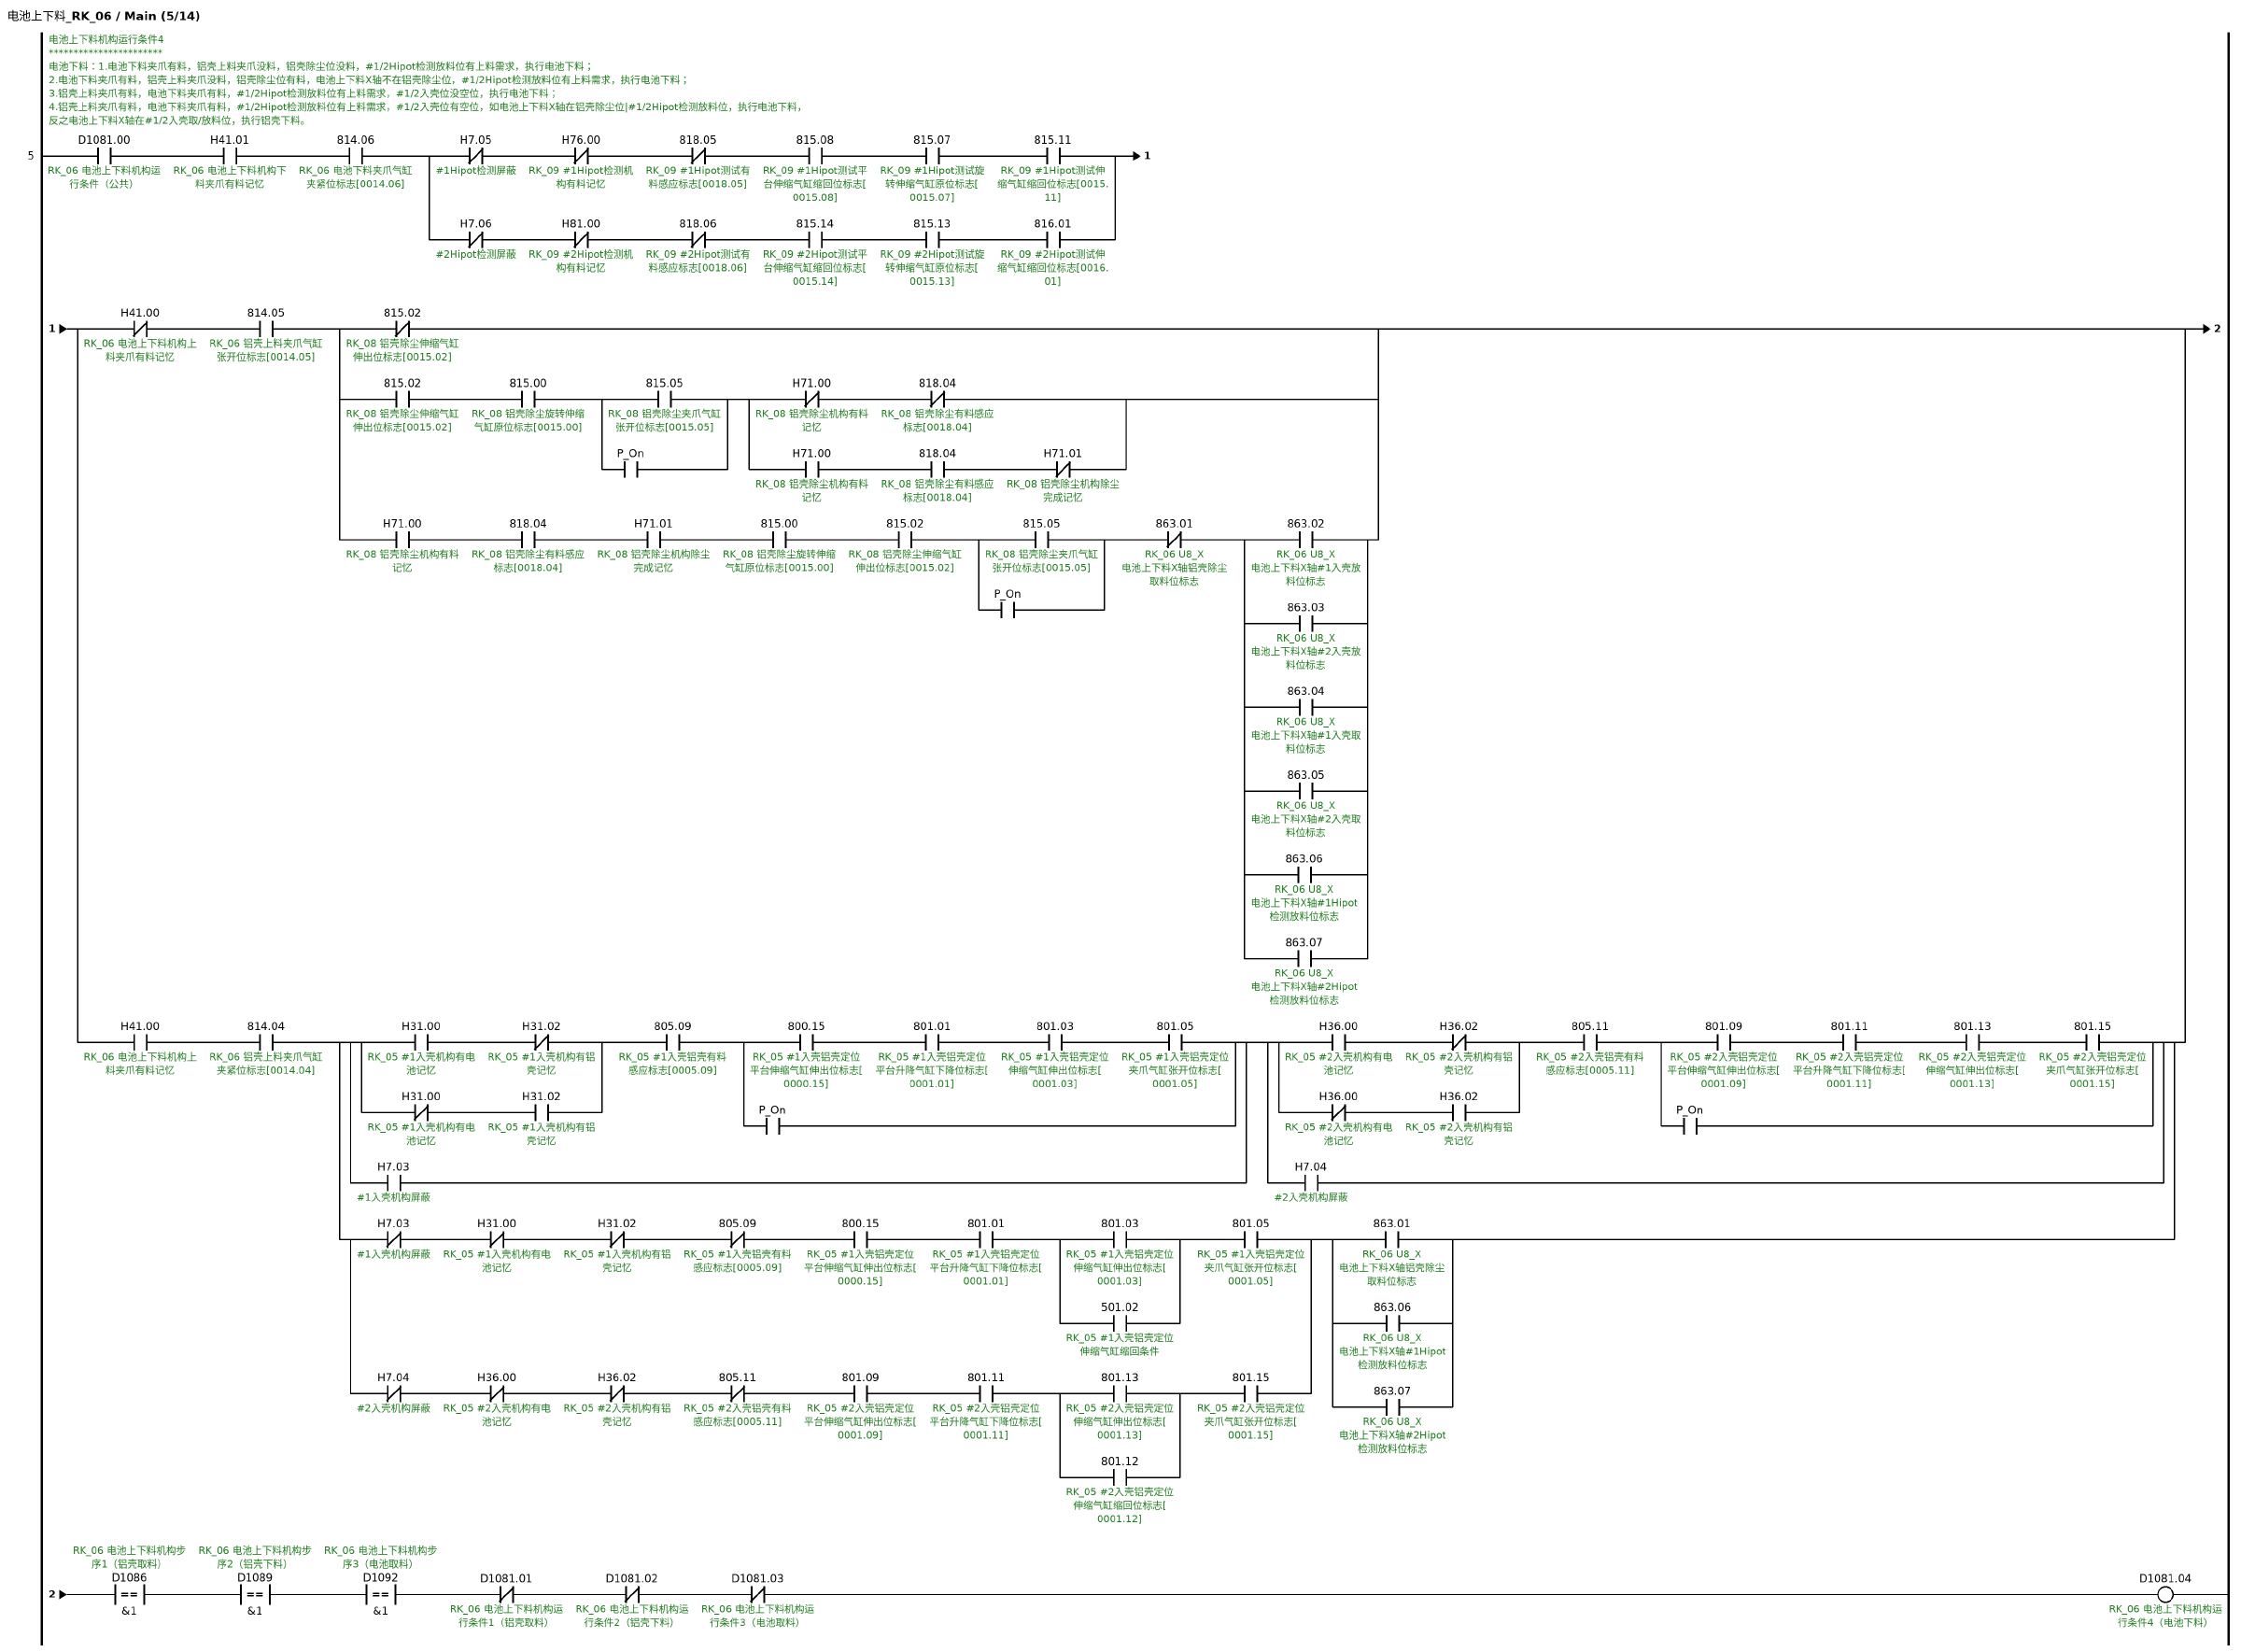
; rung 5: 电池上下料机构运行条件4 / *********************** / 电池下料：1.电池下料夹爪有料，铝壳上料夹爪没料，铝壳除尘位没料，#1/2Hipot检测放料位有上料需求，执行电池下料； / 2.电池下料夹爪有料，铝壳上料夹爪没料，铝壳除尘位有料，电池上下料X轴不在铝壳除尘位，#1/2Hipot检测放料位有上料需求，执行电池下料； / 3.铝壳上料夹爪有料，电池下料夹爪有料，#1/2Hipot检测放料位有上料需求，#1/2入壳位没空位，执行电池下料； / 4.铝壳上料夹爪有料，电池下料夹爪有料，#1/2Hipot检测放料位有上料需求，#1/2入壳位有空位，如电池上下料X轴在铝壳除尘位|#1/2Hipot检测放料位，执行电池下料， / 反之电池上下料X轴在#1/2入壳取/放料位，执行铝壳下料。
LD D1081.00  ; RK_06 电池上下料机构运行条件（公共）
AND H41.01  ; RK_06 电池上下料机构下料夹爪有料记忆
AND 814.06  ; RK_06 电池下料夹爪气缸夹紧位标志[0014.06]
LDNOT H7.05  ; #1Hipot检测屏蔽
ANDNOT H76.00  ; RK_09 #1Hipot检测机构有料记忆
ANDNOT 818.05  ; RK_09 #1Hipot测试有料感应标志[0018.05]
AND 815.08  ; RK_09 #1Hipot测试平台伸缩气缸缩回位标志[0015.08]
AND 815.07  ; RK_09 #1Hipot测试旋转伸缩气缸原位标志[0015.07]
AND 815.11  ; RK_09 #1Hipot测试伸缩气缸缩回位标志[0015.11]
LDNOT H7.06  ; #2Hipot检测屏蔽
ANDNOT H81.00  ; RK_09 #2Hipot检测机构有料记忆
ANDNOT 818.06  ; RK_09 #2Hipot测试有料感应标志[0018.06]
AND 815.14  ; RK_09 #2Hipot测试平台伸缩气缸缩回位标志[0015.14]
AND 815.13  ; RK_09 #2Hipot测试旋转伸缩气缸原位标志[0015.13]
AND 816.01  ; RK_09 #2Hipot测试伸缩气缸缩回位标志[0016.01]
ORLD
ANDLD
LDNOT H41.00  ; RK_06 电池上下料机构上料夹爪有料记忆
AND 814.05  ; RK_06 铝壳上料夹爪气缸张开位标志[0014.05]
LDNOT 815.02  ; RK_08 铝壳除尘伸缩气缸伸出位标志[0015.02]
LD 815.02  ; RK_08 铝壳除尘伸缩气缸伸出位标志[0015.02]
AND 815.00  ; RK_08 铝壳除尘旋转伸缩气缸原位标志[0015.00]
LD 815.05  ; RK_08 铝壳除尘夹爪气缸张开位标志[0015.05]
OR P_On
ANDLD
LDNOT H71.00  ; RK_08 铝壳除尘机构有料记忆
ANDNOT 818.04  ; RK_08 铝壳除尘有料感应标志[0018.04]
LD H71.00  ; RK_08 铝壳除尘机构有料记忆
AND 818.04  ; RK_08 铝壳除尘有料感应标志[0018.04]
ANDNOT H71.01  ; RK_08 铝壳除尘机构除尘完成记忆
ORLD
ANDLD
ORLD
LD H71.00  ; RK_08 铝壳除尘机构有料记忆
AND 818.04  ; RK_08 铝壳除尘有料感应标志[0018.04]
AND H71.01  ; RK_08 铝壳除尘机构除尘完成记忆
AND 815.00  ; RK_08 铝壳除尘旋转伸缩气缸原位标志[0015.00]
AND 815.02  ; RK_08 铝壳除尘伸缩气缸伸出位标志[0015.02]
LD 815.05  ; RK_08 铝壳除尘夹爪气缸张开位标志[0015.05]
OR P_On
ANDLD
ANDNOT 863.01  ; RK_06 U8_X 电池上下料X轴铝壳除尘取料位标志
LD 863.02  ; RK_06 U8_X 电池上下料X轴#1入壳放料位标志
OR 863.03  ; RK_06 U8_X 电池上下料X轴#2入壳放料位标志
OR 863.04  ; RK_06 U8_X 电池上下料X轴#1入壳取料位标志
OR 863.05  ; RK_06 U8_X 电池上下料X轴#2入壳取料位标志
OR 863.06  ; RK_06 U8_X 电池上下料X轴#1Hipot检测放料位标志
OR 863.07  ; RK_06 U8_X 电池上下料X轴#2Hipot检测放料位标志
ANDLD
ORLD
ANDLD
LD H41.00  ; RK_06 电池上下料机构上料夹爪有料记忆
AND 814.04  ; RK_06 铝壳上料夹爪气缸夹紧位标志[0014.04]
LD H31.00  ; RK_05 #1入壳机构有电池记忆
ANDNOT H31.02  ; RK_05 #1入壳机构有铝壳记忆
LDNOT H31.00  ; RK_05 #1入壳机构有电池记忆
AND H31.02  ; RK_05 #1入壳机构有铝壳记忆
ORLD
AND 805.09  ; RK_05 #1入壳铝壳有料感应标志[0005.09]
LD 800.15  ; RK_05 #1入壳铝壳定位平台伸缩气缸伸出位标志[0000.15]
AND 801.01  ; RK_05 #1入壳铝壳定位平台升降气缸下降位标志[0001.01]
AND 801.03  ; RK_05 #1入壳铝壳定位伸缩气缸伸出位标志[0001.03]
AND 801.05  ; RK_05 #1入壳铝壳定位夹爪气缸张开位标志[0001.05]
OR P_On
ANDLD
OR H7.03  ; #1入壳机构屏蔽
LD H36.00  ; RK_05 #2入壳机构有电池记忆
ANDNOT H36.02  ; RK_05 #2入壳机构有铝壳记忆
LDNOT H36.00  ; RK_05 #2入壳机构有电池记忆
AND H36.02  ; RK_05 #2入壳机构有铝壳记忆
ORLD
AND 805.11  ; RK_05 #2入壳铝壳有料感应标志[0005.11]
LD 801.09  ; RK_05 #2入壳铝壳定位平台伸缩气缸伸出位标志[0001.09]
AND 801.11  ; RK_05 #2入壳铝壳定位平台升降气缸下降位标志[0001.11]
AND 801.13  ; RK_05 #2入壳铝壳定位伸缩气缸伸出位标志[0001.13]
AND 801.15  ; RK_05 #2入壳铝壳定位夹爪气缸张开位标志[0001.15]
OR P_On
ANDLD
OR H7.04  ; #2入壳机构屏蔽
ANDLD
LDNOT H7.03  ; #1入壳机构屏蔽
ANDNOT H31.00  ; RK_05 #1入壳机构有电池记忆
ANDNOT H31.02  ; RK_05 #1入壳机构有铝壳记忆
ANDNOT 805.09  ; RK_05 #1入壳铝壳有料感应标志[0005.09]
AND 800.15  ; RK_05 #1入壳铝壳定位平台伸缩气缸伸出位标志[0000.15]
AND 801.01  ; RK_05 #1入壳铝壳定位平台升降气缸下降位标志[0001.01]
LD 801.03  ; RK_05 #1入壳铝壳定位伸缩气缸伸出位标志[0001.03]
OR 501.02  ; RK_05 #1入壳铝壳定位伸缩气缸缩回条件
ANDLD
AND 801.05  ; RK_05 #1入壳铝壳定位夹爪气缸张开位标志[0001.05]
LDNOT H7.04  ; #2入壳机构屏蔽
ANDNOT H36.00  ; RK_05 #2入壳机构有电池记忆
ANDNOT H36.02  ; RK_05 #2入壳机构有铝壳记忆
ANDNOT 805.11  ; RK_05 #2入壳铝壳有料感应标志[0005.11]
AND 801.09  ; RK_05 #2入壳铝壳定位平台伸缩气缸伸出位标志[0001.09]
AND 801.11  ; RK_05 #2入壳铝壳定位平台升降气缸下降位标志[0001.11]
LD 801.13  ; RK_05 #2入壳铝壳定位伸缩气缸伸出位标志[0001.13]
OR 801.12  ; RK_05 #2入壳铝壳定位伸缩气缸缩回位标志[0001.12]
ANDLD
AND 801.15  ; RK_05 #2入壳铝壳定位夹爪气缸张开位标志[0001.15]
ORLD
LD 863.01  ; RK_06 U8_X 电池上下料X轴铝壳除尘取料位标志
OR 863.06  ; RK_06 U8_X 电池上下料X轴#1Hipot检测放料位标志
OR 863.07  ; RK_06 U8_X 电池上下料X轴#2Hipot检测放料位标志
ANDLD
ORLD
ANDLD
ORLD
ANDLD
AND=(300) D1086 &1  ; RK_06 电池上下料机构步序1（铝壳取料）
AND=(300) D1089 &1  ; RK_06 电池上下料机构步序2（铝壳下料）
AND=(300) D1092 &1  ; RK_06 电池上下料机构步序3（电池取料）
ANDNOT D1081.01  ; RK_06 电池上下料机构运行条件1（铝壳取料）
ANDNOT D1081.02  ; RK_06 电池上下料机构运行条件2（铝壳下料）
ANDNOT D1081.03  ; RK_06 电池上下料机构运行条件3（电池取料）
OUT D1081.04  ; RK_06 电池上下料机构运行条件4（电池下料）

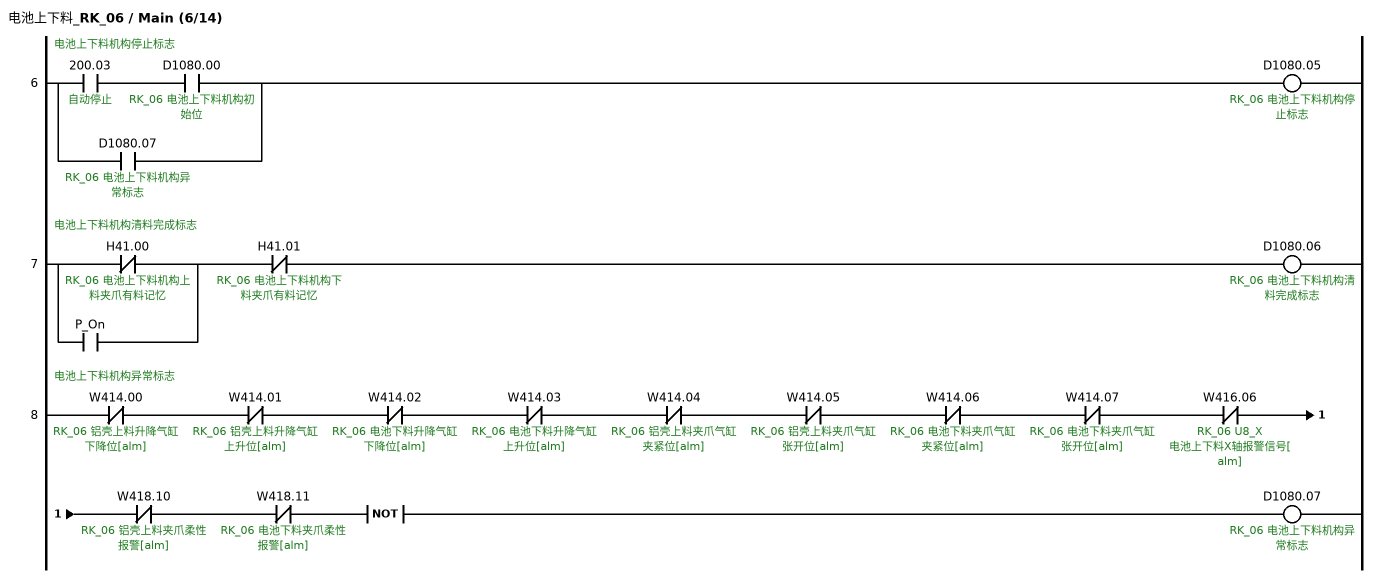
; rung 6: 电池上下料机构停止标志
LD 200.03  ; 自动停止
AND D1080.00  ; RK_06 电池上下料机构初始位
OR D1080.07  ; RK_06 电池上下料机构异常标志
OUT D1080.05  ; RK_06 电池上下料机构停止标志
; rung 7: 电池上下料机构清料完成标志
LDNOT H41.00  ; RK_06 电池上下料机构上料夹爪有料记忆
OR P_On
ANDNOT H41.01  ; RK_06 电池上下料机构下料夹爪有料记忆
OUT D1080.06  ; RK_06 电池上下料机构清料完成标志
; rung 8: 电池上下料机构异常标志
LDNOT W414.00  ; RK_06 铝壳上料升降气缸下降位[alm]
ANDNOT W414.01  ; RK_06 铝壳上料升降气缸上升位[alm]
ANDNOT W414.02  ; RK_06 电池下料升降气缸下降位[alm]
ANDNOT W414.03  ; RK_06 电池下料升降气缸上升位[alm]
ANDNOT W414.04  ; RK_06 铝壳上料夹爪气缸夹紧位[alm]
ANDNOT W414.05  ; RK_06 铝壳上料夹爪气缸张开位[alm]
ANDNOT W414.06  ; RK_06 电池下料夹爪气缸夹紧位[alm]
ANDNOT W414.07  ; RK_06 电池下料夹爪气缸张开位[alm]
ANDNOT W416.06  ; RK_06 U8_X 电池上下料X轴报警信号[alm]
ANDNOT W418.10  ; RK_06 铝壳上料夹爪柔性报警[alm]
ANDNOT W418.11  ; RK_06 电池下料夹爪柔性报警[alm]
NOT(520)
OUT D1080.07  ; RK_06 电池上下料机构异常标志

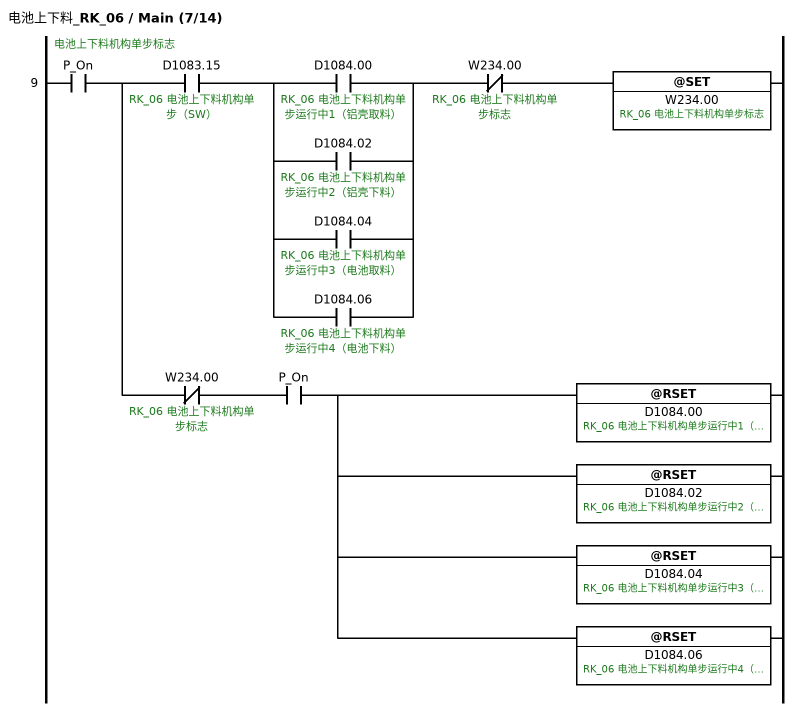
; rung 9: 电池上下料机构单步标志
LD P_On
OUT TR0
AND D1083.15  ; RK_06 电池上下料机构单步（SW）
LD D1084.00  ; RK_06 电池上下料机构单步运行中1（铝壳取料）
OR D1084.02  ; RK_06 电池上下料机构单步运行中2（铝壳下料）
OR D1084.04  ; RK_06 电池上下料机构单步运行中3（电池取料）
OR D1084.06  ; RK_06 电池上下料机构单步运行中4（电池下料）
ANDLD
ANDNOT W234.00  ; RK_06 电池上下料机构单步标志
@SET W234.00  ; RK_06 电池上下料机构单步标志
LD TR0
ANDNOT W234.00  ; RK_06 电池上下料机构单步标志
AND P_On
@RSET D1084.00  ; RK_06 电池上下料机构单步运行中1（铝壳取料）
@RSET D1084.02  ; RK_06 电池上下料机构单步运行中2（铝壳下料）
@RSET D1084.04  ; RK_06 电池上下料机构单步运行中3（电池取料）
@RSET D1084.06  ; RK_06 电池上下料机构单步运行中4（电池下料）

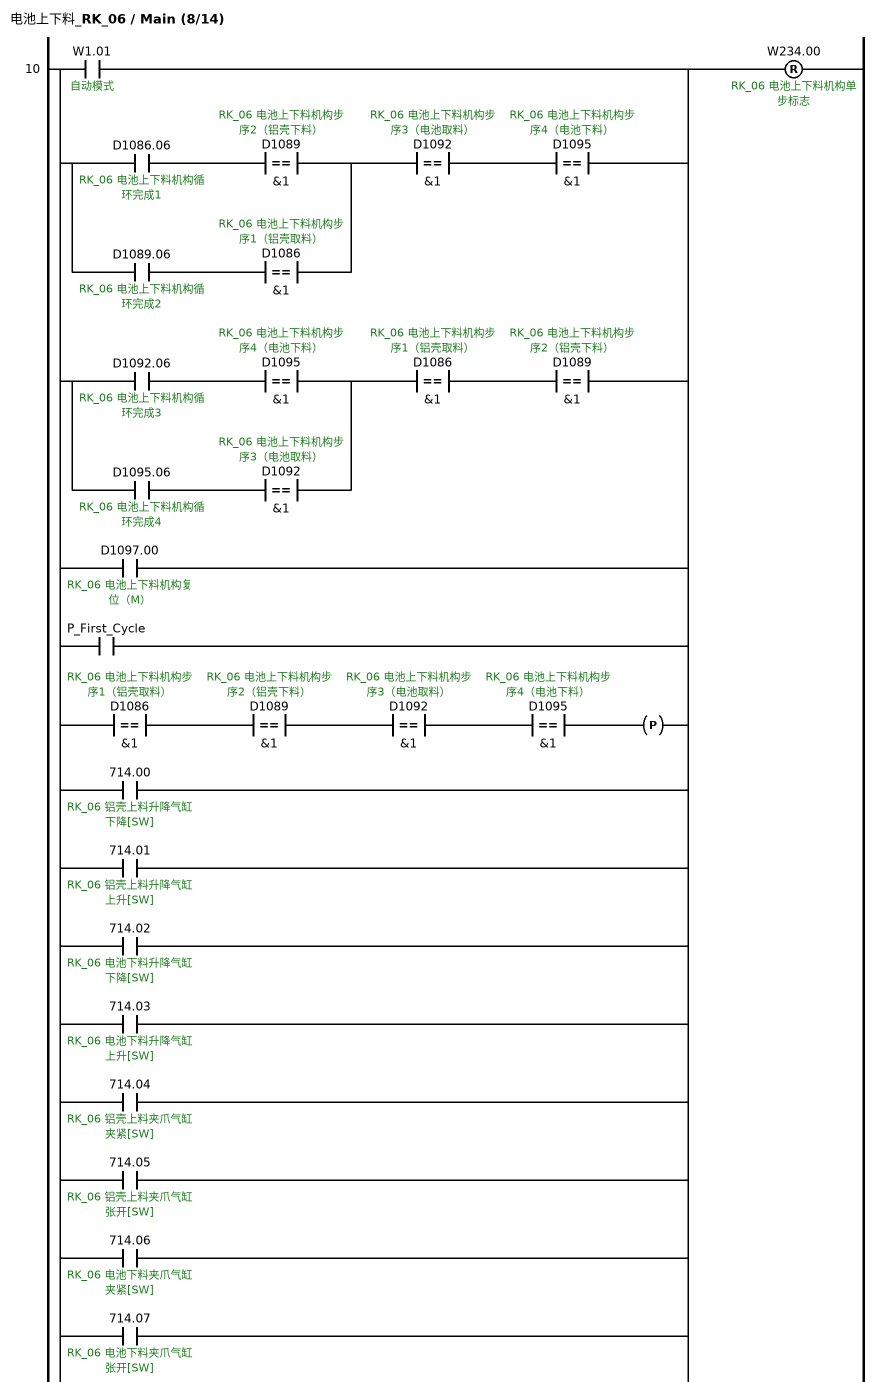

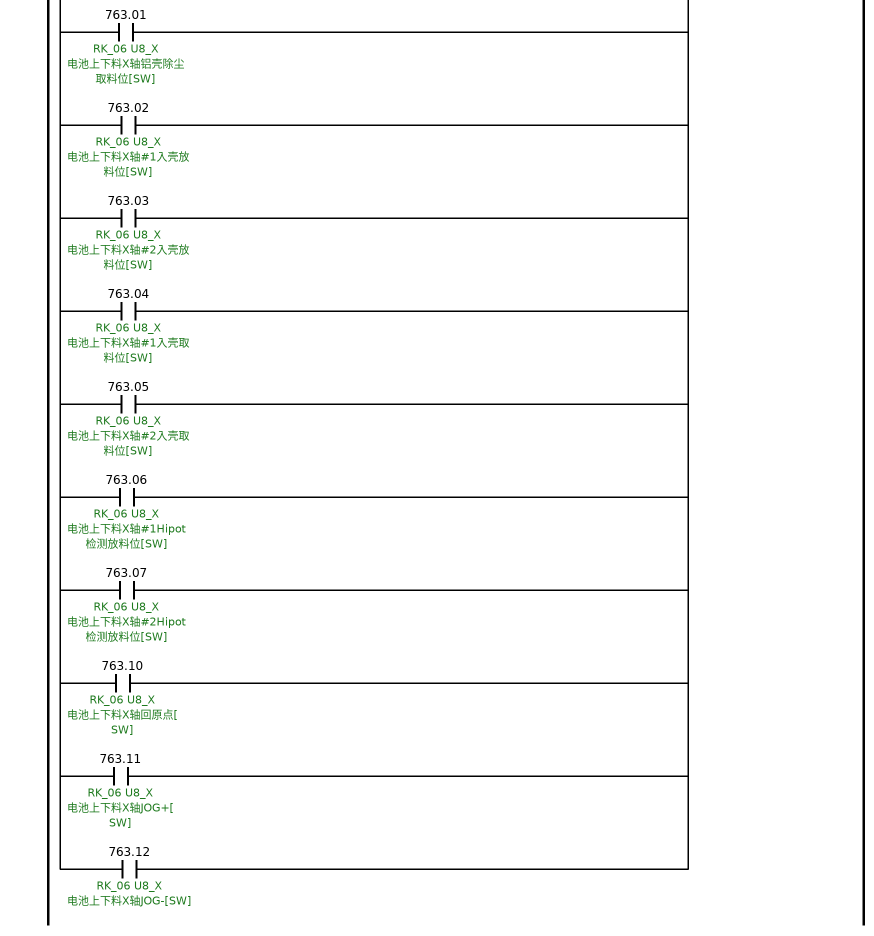
; rung 10
LD W1.01  ; 自动模式
LD D1086.06  ; RK_06 电池上下料机构循环完成1
AND=(300) D1089 &1  ; RK_06 电池上下料机构步序2（铝壳下料）
LD D1089.06  ; RK_06 电池上下料机构循环完成2
AND=(300) D1086 &1  ; RK_06 电池上下料机构步序1（铝壳取料）
ORLD
AND=(300) D1092 &1  ; RK_06 电池上下料机构步序3（电池取料）
AND=(300) D1095 &1  ; RK_06 电池上下料机构步序4（电池下料）
ORLD
LD D1092.06  ; RK_06 电池上下料机构循环完成3
AND=(300) D1095 &1  ; RK_06 电池上下料机构步序4（电池下料）
LD D1095.06  ; RK_06 电池上下料机构循环完成4
AND=(300) D1092 &1  ; RK_06 电池上下料机构步序3（电池取料）
ORLD
AND=(300) D1086 &1  ; RK_06 电池上下料机构步序1（铝壳取料）
AND=(300) D1089 &1  ; RK_06 电池上下料机构步序2（铝壳下料）
ORLD
OR D1097.00  ; RK_06 电池上下料机构复位（M）
OR P_First_Cycle
LD=(300) D1086 &1  ; RK_06 电池上下料机构步序1（铝壳取料）
AND=(300) D1089 &1  ; RK_06 电池上下料机构步序2（铝壳下料）
AND=(300) D1092 &1  ; RK_06 电池上下料机构步序3（电池取料）
AND=(300) D1095 &1  ; RK_06 电池上下料机构步序4（电池下料）
UP(521)
ORLD
OR 714.00  ; RK_06 铝壳上料升降气缸下降[SW]
OR 714.01  ; RK_06 铝壳上料升降气缸上升[SW]
OR 714.02  ; RK_06 电池下料升降气缸下降[SW]
OR 714.03  ; RK_06 电池下料升降气缸上升[SW]
OR 714.04  ; RK_06 铝壳上料夹爪气缸夹紧[SW]
OR 714.05  ; RK_06 铝壳上料夹爪气缸张开[SW]
OR 714.06  ; RK_06 电池下料夹爪气缸夹紧[SW]
OR 714.07  ; RK_06 电池下料夹爪气缸张开[SW]
OR 763.01  ; RK_06 U8_X 电池上下料X轴铝壳除尘取料位[SW]
OR 763.02  ; RK_06 U8_X 电池上下料X轴#1入壳放料位[SW]
OR 763.03  ; RK_06 U8_X 电池上下料X轴#2入壳放料位[SW]
OR 763.04  ; RK_06 U8_X 电池上下料X轴#1入壳取料位[SW]
OR 763.05  ; RK_06 U8_X 电池上下料X轴#2入壳取料位[SW]
OR 763.06  ; RK_06 U8_X 电池上下料X轴#1Hipot检测放料位[SW]
OR 763.07  ; RK_06 U8_X 电池上下料X轴#2Hipot检测放料位[SW]
LD 763.10  ; RK_06 U8_X 电池上下料X轴回原点[SW]
OR 763.11  ; RK_06 U8_X 电池上下料X轴JOG+[SW]
ORLD
OR 763.12  ; RK_06 U8_X 电池上下料X轴JOG-[SW]
RSET W234.00  ; RK_06 电池上下料机构单步标志

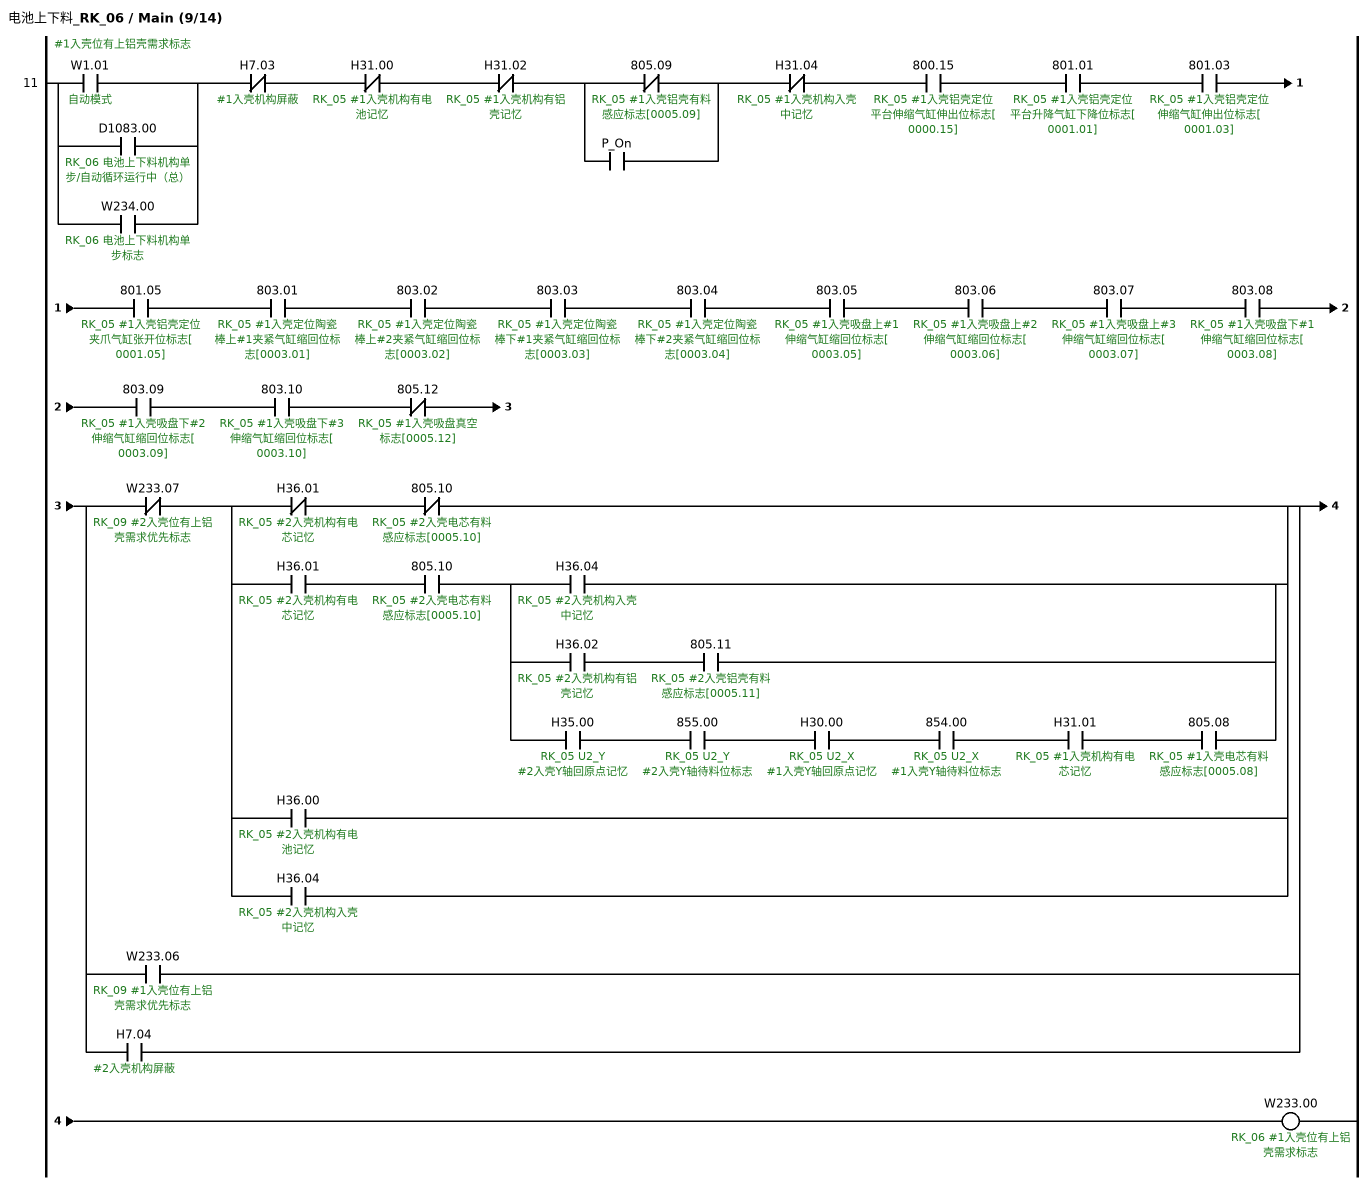
; rung 11: #1入壳位有上铝壳需求标志
LD W1.01  ; 自动模式
OR D1083.00  ; RK_06 电池上下料机构单步/自动循环运行中（总）
OR W234.00  ; RK_06 电池上下料机构单步标志
ANDNOT H7.03  ; #1入壳机构屏蔽
ANDNOT H31.00  ; RK_05 #1入壳机构有电池记忆
ANDNOT H31.02  ; RK_05 #1入壳机构有铝壳记忆
LDNOT 805.09  ; RK_05 #1入壳铝壳有料感应标志[0005.09]
OR P_On
ANDLD
ANDNOT H31.04  ; RK_05 #1入壳机构入壳中记忆
AND 800.15  ; RK_05 #1入壳铝壳定位平台伸缩气缸伸出位标志[0000.15]
AND 801.01  ; RK_05 #1入壳铝壳定位平台升降气缸下降位标志[0001.01]
AND 801.03  ; RK_05 #1入壳铝壳定位伸缩气缸伸出位标志[0001.03]
AND 801.05  ; RK_05 #1入壳铝壳定位夹爪气缸张开位标志[0001.05]
AND 803.01  ; RK_05 #1入壳定位陶瓷棒上#1夹紧气缸缩回位标志[0003.01]
AND 803.02  ; RK_05 #1入壳定位陶瓷棒上#2夹紧气缸缩回位标志[0003.02]
AND 803.03  ; RK_05 #1入壳定位陶瓷棒下#1夹紧气缸缩回位标志[0003.03]
AND 803.04  ; RK_05 #1入壳定位陶瓷棒下#2夹紧气缸缩回位标志[0003.04]
AND 803.05  ; RK_05 #1入壳吸盘上#1伸缩气缸缩回位标志[0003.05]
AND 803.06  ; RK_05 #1入壳吸盘上#2伸缩气缸缩回位标志[0003.06]
AND 803.07  ; RK_05 #1入壳吸盘上#3伸缩气缸缩回位标志[0003.07]
AND 803.08  ; RK_05 #1入壳吸盘下#1伸缩气缸缩回位标志[0003.08]
AND 803.09  ; RK_05 #1入壳吸盘下#2伸缩气缸缩回位标志[0003.09]
AND 803.10  ; RK_05 #1入壳吸盘下#3伸缩气缸缩回位标志[0003.10]
ANDNOT 805.12  ; RK_05 #1入壳吸盘真空标志[0005.12]
LDNOT W233.07  ; RK_09 #2入壳位有上铝壳需求优先标志
LDNOT H36.01  ; RK_05 #2入壳机构有电芯记忆
ANDNOT 805.10  ; RK_05 #2入壳电芯有料感应标志[0005.10]
LD H36.01  ; RK_05 #2入壳机构有电芯记忆
AND 805.10  ; RK_05 #2入壳电芯有料感应标志[0005.10]
LD H36.04  ; RK_05 #2入壳机构入壳中记忆
LD H36.02  ; RK_05 #2入壳机构有铝壳记忆
AND 805.11  ; RK_05 #2入壳铝壳有料感应标志[0005.11]
ORLD
LD H35.00  ; RK_05 U2_Y #2入壳Y轴回原点记忆
AND 855.00  ; RK_05 U2_Y #2入壳Y轴待料位标志
AND H30.00  ; RK_05 U2_X #1入壳Y轴回原点记忆
AND 854.00  ; RK_05 U2_X #1入壳Y轴待料位标志
AND H31.01  ; RK_05 #1入壳机构有电芯记忆
AND 805.08  ; RK_05 #1入壳电芯有料感应标志[0005.08]
ORLD
ANDLD
ORLD
OR H36.00  ; RK_05 #2入壳机构有电池记忆
OR H36.04  ; RK_05 #2入壳机构入壳中记忆
ANDLD
OR W233.06  ; RK_09 #1入壳位有上铝壳需求优先标志
OR H7.04  ; #2入壳机构屏蔽
ANDLD
OUT W233.00  ; RK_06 #1入壳位有上铝壳需求标志

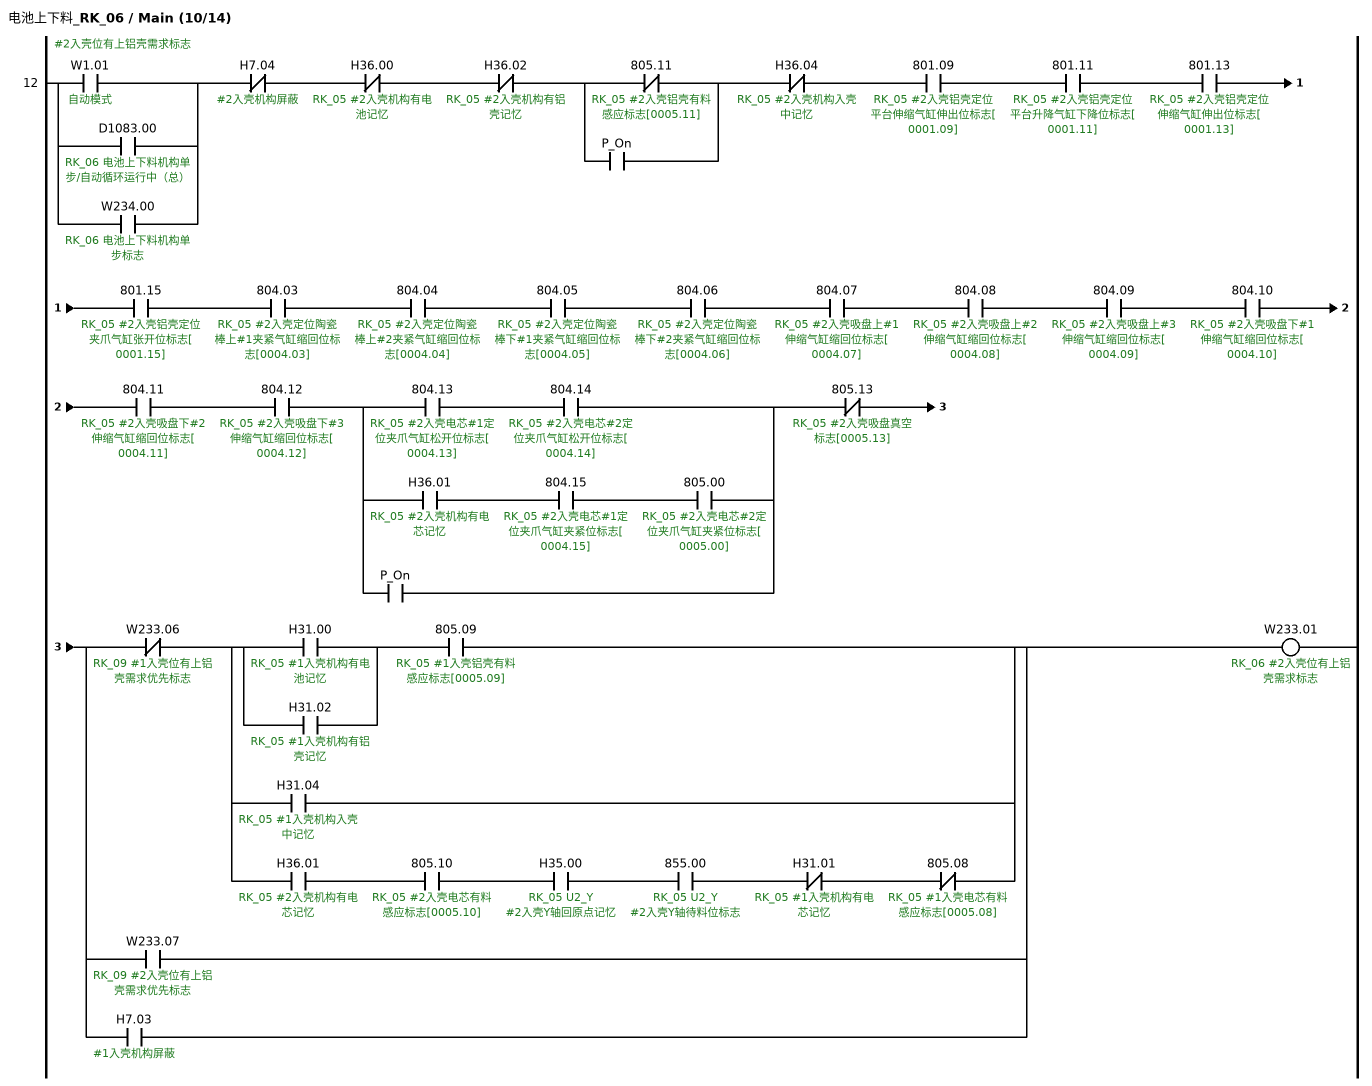
; rung 12: #2入壳位有上铝壳需求标志
LD W1.01  ; 自动模式
OR D1083.00  ; RK_06 电池上下料机构单步/自动循环运行中（总）
OR W234.00  ; RK_06 电池上下料机构单步标志
ANDNOT H7.04  ; #2入壳机构屏蔽
ANDNOT H36.00  ; RK_05 #2入壳机构有电池记忆
ANDNOT H36.02  ; RK_05 #2入壳机构有铝壳记忆
LDNOT 805.11  ; RK_05 #2入壳铝壳有料感应标志[0005.11]
OR P_On
ANDLD
ANDNOT H36.04  ; RK_05 #2入壳机构入壳中记忆
AND 801.09  ; RK_05 #2入壳铝壳定位平台伸缩气缸伸出位标志[0001.09]
AND 801.11  ; RK_05 #2入壳铝壳定位平台升降气缸下降位标志[0001.11]
AND 801.13  ; RK_05 #2入壳铝壳定位伸缩气缸伸出位标志[0001.13]
AND 801.15  ; RK_05 #2入壳铝壳定位夹爪气缸张开位标志[0001.15]
AND 804.03  ; RK_05 #2入壳定位陶瓷棒上#1夹紧气缸缩回位标志[0004.03]
AND 804.04  ; RK_05 #2入壳定位陶瓷棒上#2夹紧气缸缩回位标志[0004.04]
AND 804.05  ; RK_05 #2入壳定位陶瓷棒下#1夹紧气缸缩回位标志[0004.05]
AND 804.06  ; RK_05 #2入壳定位陶瓷棒下#2夹紧气缸缩回位标志[0004.06]
AND 804.07  ; RK_05 #2入壳吸盘上#1伸缩气缸缩回位标志[0004.07]
AND 804.08  ; RK_05 #2入壳吸盘上#2伸缩气缸缩回位标志[0004.08]
AND 804.09  ; RK_05 #2入壳吸盘上#3伸缩气缸缩回位标志[0004.09]
AND 804.10  ; RK_05 #2入壳吸盘下#1伸缩气缸缩回位标志[0004.10]
AND 804.11  ; RK_05 #2入壳吸盘下#2伸缩气缸缩回位标志[0004.11]
AND 804.12  ; RK_05 #2入壳吸盘下#3伸缩气缸缩回位标志[0004.12]
LD 804.13  ; RK_05 #2入壳电芯#1定位夹爪气缸松开位标志[0004.13]
AND 804.14  ; RK_05 #2入壳电芯#2定位夹爪气缸松开位标志[0004.14]
LD H36.01  ; RK_05 #2入壳机构有电芯记忆
AND 804.15  ; RK_05 #2入壳电芯#1定位夹爪气缸夹紧位标志[0004.15]
AND 805.00  ; RK_05 #2入壳电芯#2定位夹爪气缸夹紧位标志[0005.00]
ORLD
OR P_On
ANDLD
ANDNOT 805.13  ; RK_05 #2入壳吸盘真空标志[0005.13]
LDNOT W233.06  ; RK_09 #1入壳位有上铝壳需求优先标志
LD H31.00  ; RK_05 #1入壳机构有电池记忆
OR H31.02  ; RK_05 #1入壳机构有铝壳记忆
AND 805.09  ; RK_05 #1入壳铝壳有料感应标志[0005.09]
OR H31.04  ; RK_05 #1入壳机构入壳中记忆
LD H36.01  ; RK_05 #2入壳机构有电芯记忆
AND 805.10  ; RK_05 #2入壳电芯有料感应标志[0005.10]
AND H35.00  ; RK_05 U2_Y #2入壳Y轴回原点记忆
AND 855.00  ; RK_05 U2_Y #2入壳Y轴待料位标志
ANDNOT H31.01  ; RK_05 #1入壳机构有电芯记忆
ANDNOT 805.08  ; RK_05 #1入壳电芯有料感应标志[0005.08]
ORLD
ANDLD
OR W233.07  ; RK_09 #2入壳位有上铝壳需求优先标志
OR H7.03  ; #1入壳机构屏蔽
ANDLD
OUT W233.01  ; RK_06 #2入壳位有上铝壳需求标志

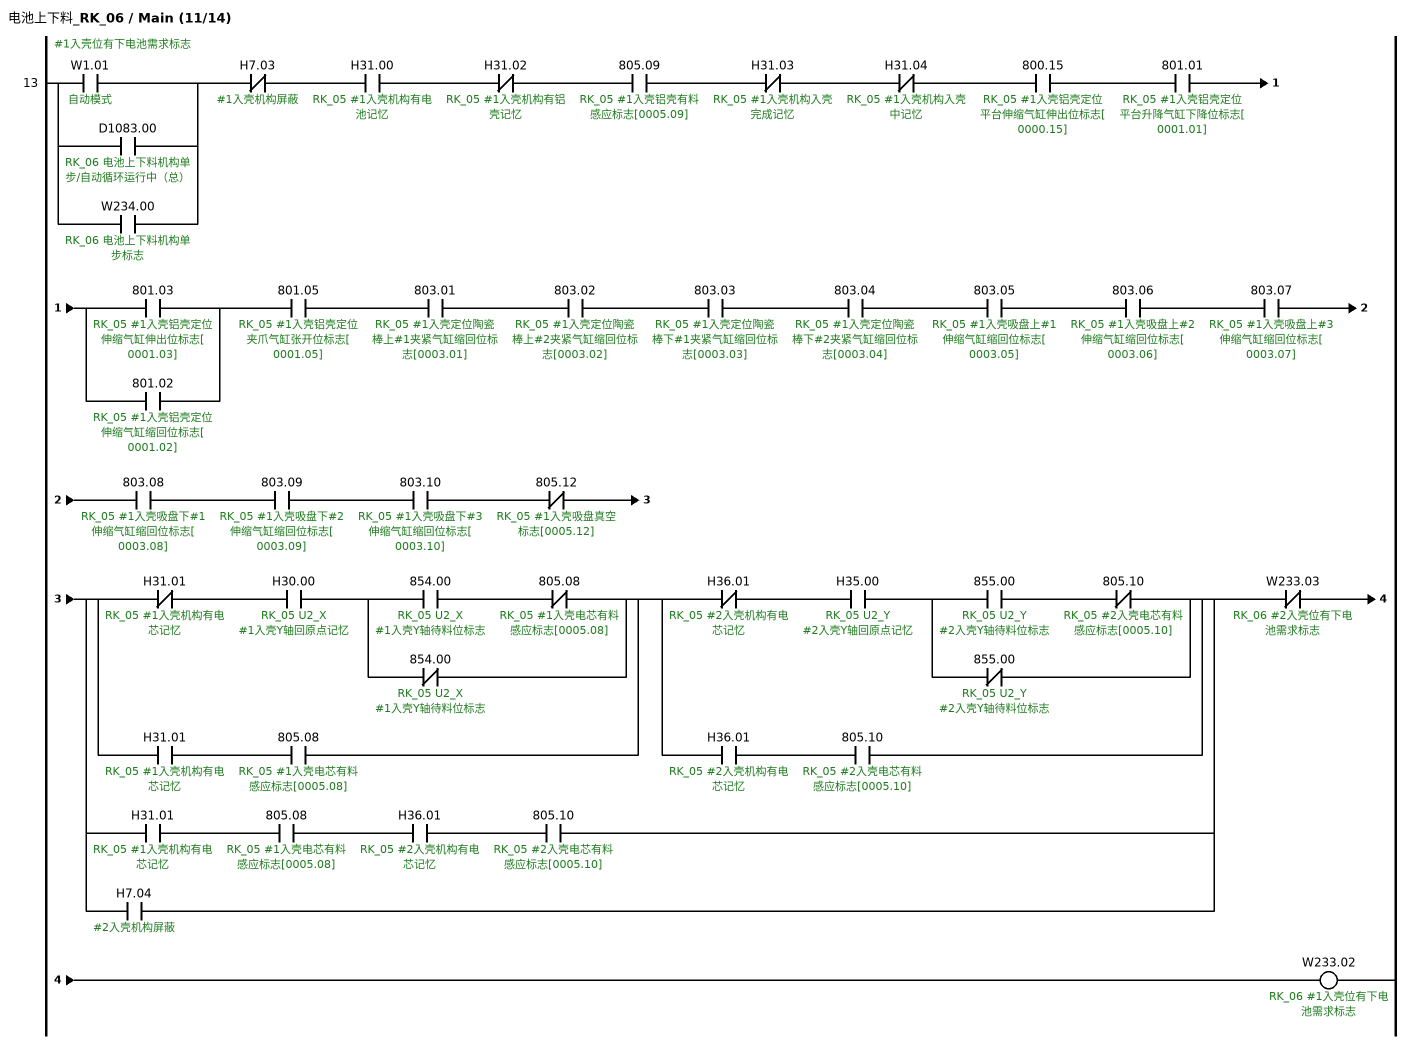
; rung 13: #1入壳位有下电池需求标志
LD W1.01  ; 自动模式
OR D1083.00  ; RK_06 电池上下料机构单步/自动循环运行中（总）
OR W234.00  ; RK_06 电池上下料机构单步标志
ANDNOT H7.03  ; #1入壳机构屏蔽
AND H31.00  ; RK_05 #1入壳机构有电池记忆
ANDNOT H31.02  ; RK_05 #1入壳机构有铝壳记忆
AND 805.09  ; RK_05 #1入壳铝壳有料感应标志[0005.09]
ANDNOT H31.03  ; RK_05 #1入壳机构入壳完成记忆
ANDNOT H31.04  ; RK_05 #1入壳机构入壳中记忆
AND 800.15  ; RK_05 #1入壳铝壳定位平台伸缩气缸伸出位标志[0000.15]
AND 801.01  ; RK_05 #1入壳铝壳定位平台升降气缸下降位标志[0001.01]
LD 801.03  ; RK_05 #1入壳铝壳定位伸缩气缸伸出位标志[0001.03]
OR 801.02  ; RK_05 #1入壳铝壳定位伸缩气缸缩回位标志[0001.02]
ANDLD
AND 801.05  ; RK_05 #1入壳铝壳定位夹爪气缸张开位标志[0001.05]
AND 803.01  ; RK_05 #1入壳定位陶瓷棒上#1夹紧气缸缩回位标志[0003.01]
AND 803.02  ; RK_05 #1入壳定位陶瓷棒上#2夹紧气缸缩回位标志[0003.02]
AND 803.03  ; RK_05 #1入壳定位陶瓷棒下#1夹紧气缸缩回位标志[0003.03]
AND 803.04  ; RK_05 #1入壳定位陶瓷棒下#2夹紧气缸缩回位标志[0003.04]
AND 803.05  ; RK_05 #1入壳吸盘上#1伸缩气缸缩回位标志[0003.05]
AND 803.06  ; RK_05 #1入壳吸盘上#2伸缩气缸缩回位标志[0003.06]
AND 803.07  ; RK_05 #1入壳吸盘上#3伸缩气缸缩回位标志[0003.07]
AND 803.08  ; RK_05 #1入壳吸盘下#1伸缩气缸缩回位标志[0003.08]
AND 803.09  ; RK_05 #1入壳吸盘下#2伸缩气缸缩回位标志[0003.09]
AND 803.10  ; RK_05 #1入壳吸盘下#3伸缩气缸缩回位标志[0003.10]
ANDNOT 805.12  ; RK_05 #1入壳吸盘真空标志[0005.12]
LDNOT H31.01  ; RK_05 #1入壳机构有电芯记忆
AND H30.00  ; RK_05 U2_X #1入壳Y轴回原点记忆
LD 854.00  ; RK_05 U2_X #1入壳Y轴待料位标志
ANDNOT 805.08  ; RK_05 #1入壳电芯有料感应标志[0005.08]
ORNOT 854.00  ; RK_05 U2_X #1入壳Y轴待料位标志
ANDLD
LD H31.01  ; RK_05 #1入壳机构有电芯记忆
AND 805.08  ; RK_05 #1入壳电芯有料感应标志[0005.08]
ORLD
LDNOT H36.01  ; RK_05 #2入壳机构有电芯记忆
AND H35.00  ; RK_05 U2_Y #2入壳Y轴回原点记忆
LD 855.00  ; RK_05 U2_Y #2入壳Y轴待料位标志
ANDNOT 805.10  ; RK_05 #2入壳电芯有料感应标志[0005.10]
ORNOT 855.00  ; RK_05 U2_Y #2入壳Y轴待料位标志
ANDLD
LD H36.01  ; RK_05 #2入壳机构有电芯记忆
AND 805.10  ; RK_05 #2入壳电芯有料感应标志[0005.10]
ORLD
ANDLD
LD H31.01  ; RK_05 #1入壳机构有电芯记忆
AND 805.08  ; RK_05 #1入壳电芯有料感应标志[0005.08]
AND H36.01  ; RK_05 #2入壳机构有电芯记忆
AND 805.10  ; RK_05 #2入壳电芯有料感应标志[0005.10]
ORLD
OR H7.04  ; #2入壳机构屏蔽
ANDLD
ANDNOT W233.03  ; RK_06 #2入壳位有下电池需求标志
OUT W233.02  ; RK_06 #1入壳位有下电池需求标志

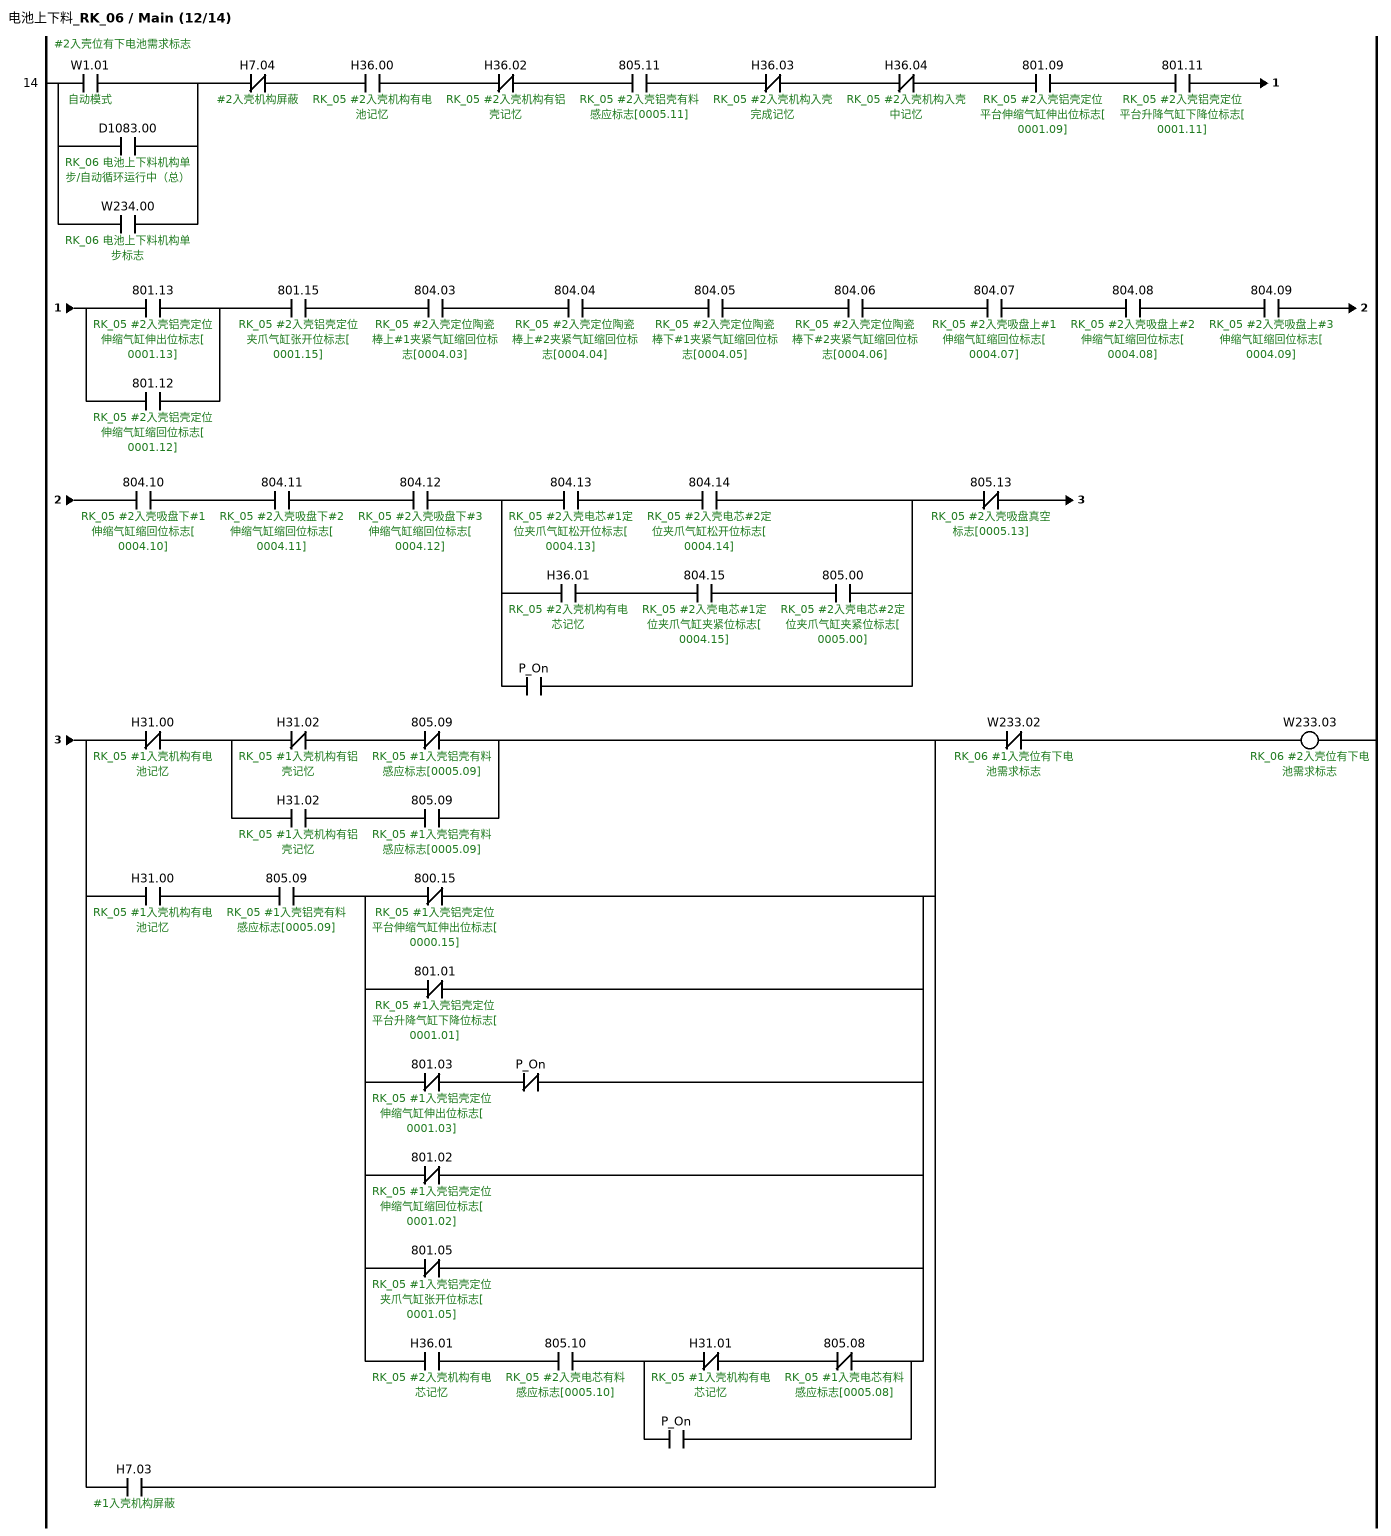
; rung 14: #2入壳位有下电池需求标志
LD W1.01  ; 自动模式
OR D1083.00  ; RK_06 电池上下料机构单步/自动循环运行中（总）
OR W234.00  ; RK_06 电池上下料机构单步标志
ANDNOT H7.04  ; #2入壳机构屏蔽
AND H36.00  ; RK_05 #2入壳机构有电池记忆
ANDNOT H36.02  ; RK_05 #2入壳机构有铝壳记忆
AND 805.11  ; RK_05 #2入壳铝壳有料感应标志[0005.11]
ANDNOT H36.03  ; RK_05 #2入壳机构入壳完成记忆
ANDNOT H36.04  ; RK_05 #2入壳机构入壳中记忆
AND 801.09  ; RK_05 #2入壳铝壳定位平台伸缩气缸伸出位标志[0001.09]
AND 801.11  ; RK_05 #2入壳铝壳定位平台升降气缸下降位标志[0001.11]
LD 801.13  ; RK_05 #2入壳铝壳定位伸缩气缸伸出位标志[0001.13]
OR 801.12  ; RK_05 #2入壳铝壳定位伸缩气缸缩回位标志[0001.12]
ANDLD
AND 801.15  ; RK_05 #2入壳铝壳定位夹爪气缸张开位标志[0001.15]
AND 804.03  ; RK_05 #2入壳定位陶瓷棒上#1夹紧气缸缩回位标志[0004.03]
AND 804.04  ; RK_05 #2入壳定位陶瓷棒上#2夹紧气缸缩回位标志[0004.04]
AND 804.05  ; RK_05 #2入壳定位陶瓷棒下#1夹紧气缸缩回位标志[0004.05]
AND 804.06  ; RK_05 #2入壳定位陶瓷棒下#2夹紧气缸缩回位标志[0004.06]
AND 804.07  ; RK_05 #2入壳吸盘上#1伸缩气缸缩回位标志[0004.07]
AND 804.08  ; RK_05 #2入壳吸盘上#2伸缩气缸缩回位标志[0004.08]
AND 804.09  ; RK_05 #2入壳吸盘上#3伸缩气缸缩回位标志[0004.09]
AND 804.10  ; RK_05 #2入壳吸盘下#1伸缩气缸缩回位标志[0004.10]
AND 804.11  ; RK_05 #2入壳吸盘下#2伸缩气缸缩回位标志[0004.11]
AND 804.12  ; RK_05 #2入壳吸盘下#3伸缩气缸缩回位标志[0004.12]
LD 804.13  ; RK_05 #2入壳电芯#1定位夹爪气缸松开位标志[0004.13]
AND 804.14  ; RK_05 #2入壳电芯#2定位夹爪气缸松开位标志[0004.14]
LD H36.01  ; RK_05 #2入壳机构有电芯记忆
AND 804.15  ; RK_05 #2入壳电芯#1定位夹爪气缸夹紧位标志[0004.15]
AND 805.00  ; RK_05 #2入壳电芯#2定位夹爪气缸夹紧位标志[0005.00]
ORLD
OR P_On
ANDLD
ANDNOT 805.13  ; RK_05 #2入壳吸盘真空标志[0005.13]
LDNOT H31.00  ; RK_05 #1入壳机构有电池记忆
LDNOT H31.02  ; RK_05 #1入壳机构有铝壳记忆
ANDNOT 805.09  ; RK_05 #1入壳铝壳有料感应标志[0005.09]
LD H31.02  ; RK_05 #1入壳机构有铝壳记忆
AND 805.09  ; RK_05 #1入壳铝壳有料感应标志[0005.09]
ORLD
ANDLD
LD H31.00  ; RK_05 #1入壳机构有电池记忆
AND 805.09  ; RK_05 #1入壳铝壳有料感应标志[0005.09]
LDNOT 800.15  ; RK_05 #1入壳铝壳定位平台伸缩气缸伸出位标志[0000.15]
ORNOT 801.01  ; RK_05 #1入壳铝壳定位平台升降气缸下降位标志[0001.01]
LDNOT 801.03  ; RK_05 #1入壳铝壳定位伸缩气缸伸出位标志[0001.03]
ANDNOT P_On
ORLD
ORNOT 801.02  ; RK_05 #1入壳铝壳定位伸缩气缸缩回位标志[0001.02]
ORNOT 801.05  ; RK_05 #1入壳铝壳定位夹爪气缸张开位标志[0001.05]
LD H36.01  ; RK_05 #2入壳机构有电芯记忆
AND 805.10  ; RK_05 #2入壳电芯有料感应标志[0005.10]
LDNOT H31.01  ; RK_05 #1入壳机构有电芯记忆
ANDNOT 805.08  ; RK_05 #1入壳电芯有料感应标志[0005.08]
OR P_On
ANDLD
ORLD
ANDLD
ORLD
OR H7.03  ; #1入壳机构屏蔽
ANDLD
ANDNOT W233.02  ; RK_06 #1入壳位有下电池需求标志
OUT W233.03  ; RK_06 #2入壳位有下电池需求标志

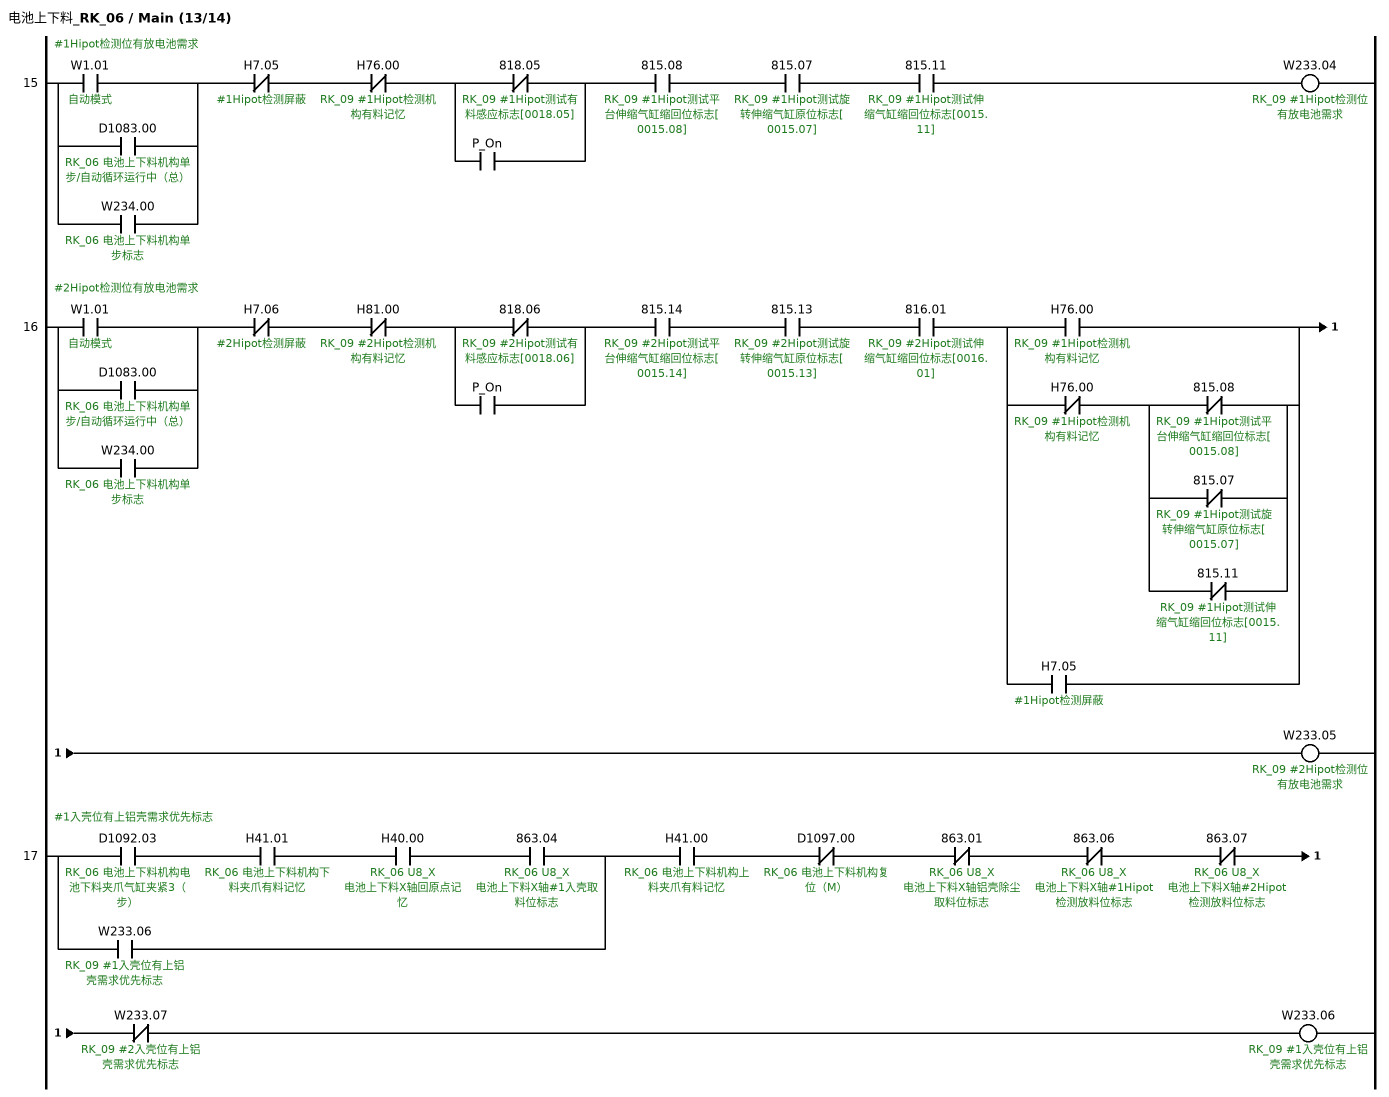
; rung 15: #1Hipot检测位有放电池需求
LD W1.01  ; 自动模式
OR D1083.00  ; RK_06 电池上下料机构单步/自动循环运行中（总）
OR W234.00  ; RK_06 电池上下料机构单步标志
ANDNOT H7.05  ; #1Hipot检测屏蔽
ANDNOT H76.00  ; RK_09 #1Hipot检测机构有料记忆
LDNOT 818.05  ; RK_09 #1Hipot测试有料感应标志[0018.05]
OR P_On
ANDLD
AND 815.08  ; RK_09 #1Hipot测试平台伸缩气缸缩回位标志[0015.08]
AND 815.07  ; RK_09 #1Hipot测试旋转伸缩气缸原位标志[0015.07]
AND 815.11  ; RK_09 #1Hipot测试伸缩气缸缩回位标志[0015.11]
OUT W233.04  ; RK_09 #1Hipot检测位有放电池需求
; rung 16: #2Hipot检测位有放电池需求
LD W1.01  ; 自动模式
OR D1083.00  ; RK_06 电池上下料机构单步/自动循环运行中（总）
OR W234.00  ; RK_06 电池上下料机构单步标志
ANDNOT H7.06  ; #2Hipot检测屏蔽
ANDNOT H81.00  ; RK_09 #2Hipot检测机构有料记忆
LDNOT 818.06  ; RK_09 #2Hipot测试有料感应标志[0018.06]
OR P_On
ANDLD
AND 815.14  ; RK_09 #2Hipot测试平台伸缩气缸缩回位标志[0015.14]
AND 815.13  ; RK_09 #2Hipot测试旋转伸缩气缸原位标志[0015.13]
AND 816.01  ; RK_09 #2Hipot测试伸缩气缸缩回位标志[0016.01]
LD H76.00  ; RK_09 #1Hipot检测机构有料记忆
LDNOT H76.00  ; RK_09 #1Hipot检测机构有料记忆
LDNOT 815.08  ; RK_09 #1Hipot测试平台伸缩气缸缩回位标志[0015.08]
ORNOT 815.07  ; RK_09 #1Hipot测试旋转伸缩气缸原位标志[0015.07]
ORNOT 815.11  ; RK_09 #1Hipot测试伸缩气缸缩回位标志[0015.11]
ANDLD
ORLD
OR H7.05  ; #1Hipot检测屏蔽
ANDLD
OUT W233.05  ; RK_09 #2Hipot检测位有放电池需求
; rung 17: #1入壳位有上铝壳需求优先标志
LD D1092.03  ; RK_06 电池上下料机构电池下料夹爪气缸夹紧3（步）
AND H41.01  ; RK_06 电池上下料机构下料夹爪有料记忆
AND H40.00  ; RK_06 U8_X 电池上下料X轴回原点记忆
AND 863.04  ; RK_06 U8_X 电池上下料X轴#1入壳取料位标志
OR W233.06  ; RK_09 #1入壳位有上铝壳需求优先标志
AND H41.00  ; RK_06 电池上下料机构上料夹爪有料记忆
ANDNOT D1097.00  ; RK_06 电池上下料机构复位（M）
ANDNOT 863.01  ; RK_06 U8_X 电池上下料X轴铝壳除尘取料位标志
ANDNOT 863.06  ; RK_06 U8_X 电池上下料X轴#1Hipot检测放料位标志
ANDNOT 863.07  ; RK_06 U8_X 电池上下料X轴#2Hipot检测放料位标志
ANDNOT W233.07  ; RK_09 #2入壳位有上铝壳需求优先标志
OUT W233.06  ; RK_09 #1入壳位有上铝壳需求优先标志  // 电池上下料机构上料夹爪有料，在电池上下料X轴#1入壳取料完成后，优先#1入壳放料！工站初始化之后优先标志取消，工站随机选择工况运行！

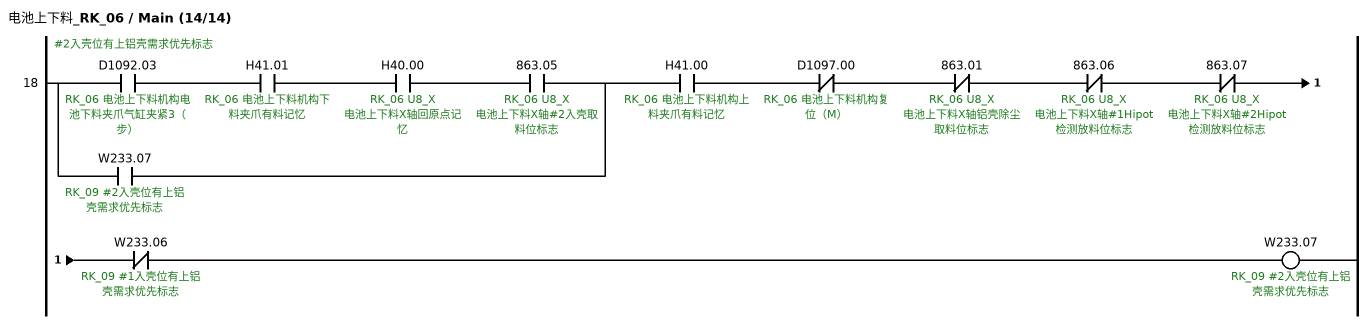
; rung 18: #2入壳位有上铝壳需求优先标志
LD D1092.03  ; RK_06 电池上下料机构电池下料夹爪气缸夹紧3（步）
AND H41.01  ; RK_06 电池上下料机构下料夹爪有料记忆
AND H40.00  ; RK_06 U8_X 电池上下料X轴回原点记忆
AND 863.05  ; RK_06 U8_X 电池上下料X轴#2入壳取料位标志
OR W233.07  ; RK_09 #2入壳位有上铝壳需求优先标志
AND H41.00  ; RK_06 电池上下料机构上料夹爪有料记忆
ANDNOT D1097.00  ; RK_06 电池上下料机构复位（M）
ANDNOT 863.01  ; RK_06 U8_X 电池上下料X轴铝壳除尘取料位标志
ANDNOT 863.06  ; RK_06 U8_X 电池上下料X轴#1Hipot检测放料位标志
ANDNOT 863.07  ; RK_06 U8_X 电池上下料X轴#2Hipot检测放料位标志
ANDNOT W233.06  ; RK_09 #1入壳位有上铝壳需求优先标志
OUT W233.07  ; RK_09 #2入壳位有上铝壳需求优先标志  // 电池上下料机构上料夹爪有料，在电池上下料X轴#2入壳取料完成后，优先#2入壳放料！工站初始化之后优先标志取消，工站随机选择工况运行！

### Section 手动

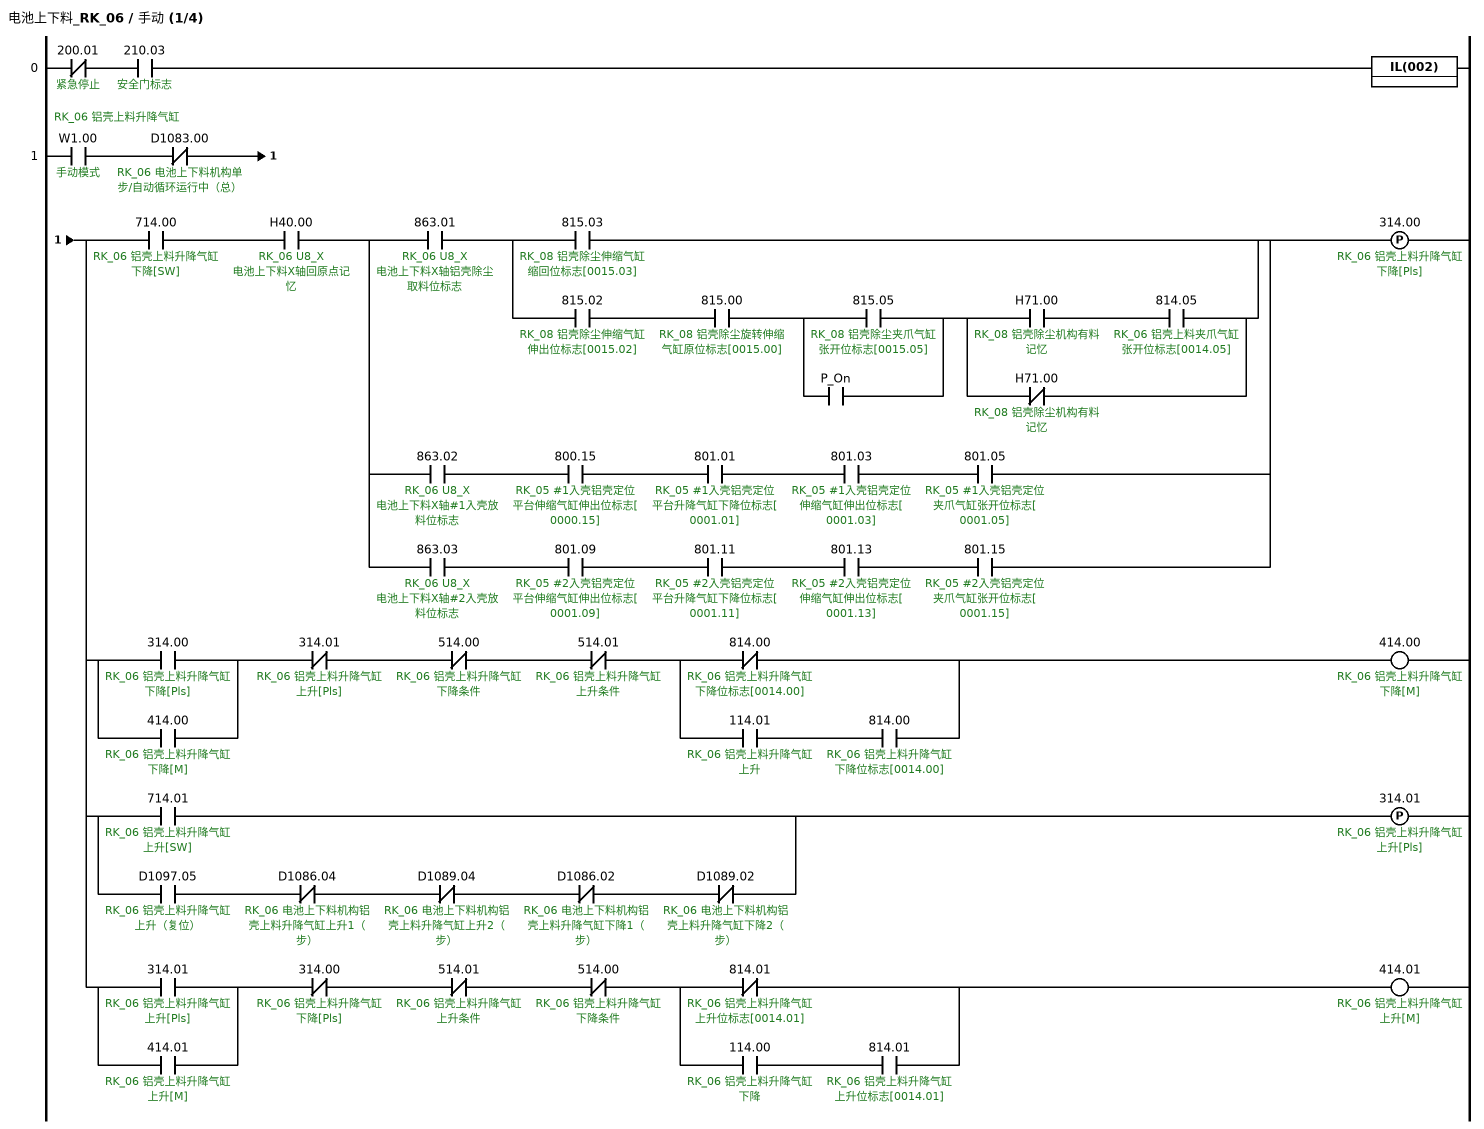
; rung 0
LDNOT 200.01  ; 紧急停止
AND 210.03  ; 安全门标志
IL(002)
; rung 1: RK_06 铝壳上料升降气缸
LD W1.00  ; 手动模式
ANDNOT D1083.00  ; RK_06 电池上下料机构单步/自动循环运行中（总）
OUT TR0
AND 714.00  ; RK_06 铝壳上料升降气缸下降[SW]
AND H40.00  ; RK_06 U8_X 电池上下料X轴回原点记忆
LD 863.01  ; RK_06 U8_X 电池上下料X轴铝壳除尘取料位标志
LD 815.03  ; RK_08 铝壳除尘伸缩气缸缩回位标志[0015.03]
LD 815.02  ; RK_08 铝壳除尘伸缩气缸伸出位标志[0015.02]
AND 815.00  ; RK_08 铝壳除尘旋转伸缩气缸原位标志[0015.00]
LD 815.05  ; RK_08 铝壳除尘夹爪气缸张开位标志[0015.05]
OR P_On
ANDLD
LD H71.00  ; RK_08 铝壳除尘机构有料记忆
AND 814.05  ; RK_06 铝壳上料夹爪气缸张开位标志[0014.05]
ORNOT H71.00  ; RK_08 铝壳除尘机构有料记忆
ANDLD
ORLD
ANDLD
LD 863.02  ; RK_06 U8_X 电池上下料X轴#1入壳放料位标志
AND 800.15  ; RK_05 #1入壳铝壳定位平台伸缩气缸伸出位标志[0000.15]
AND 801.01  ; RK_05 #1入壳铝壳定位平台升降气缸下降位标志[0001.01]
AND 801.03  ; RK_05 #1入壳铝壳定位伸缩气缸伸出位标志[0001.03]
AND 801.05  ; RK_05 #1入壳铝壳定位夹爪气缸张开位标志[0001.05]
ORLD
LD 863.03  ; RK_06 U8_X 电池上下料X轴#2入壳放料位标志
AND 801.09  ; RK_05 #2入壳铝壳定位平台伸缩气缸伸出位标志[0001.09]
AND 801.11  ; RK_05 #2入壳铝壳定位平台升降气缸下降位标志[0001.11]
AND 801.13  ; RK_05 #2入壳铝壳定位伸缩气缸伸出位标志[0001.13]
AND 801.15  ; RK_05 #2入壳铝壳定位夹爪气缸张开位标志[0001.15]
ORLD
ANDLD
DIFU(013) 314.00  ; RK_06 铝壳上料升降气缸下降[Pls]
LD TR0
LD 314.00  ; RK_06 铝壳上料升降气缸下降[Pls]
OR 414.00  ; RK_06 铝壳上料升降气缸下降[M]
ANDLD
ANDNOT 314.01  ; RK_06 铝壳上料升降气缸上升[Pls]
ANDNOT 514.00  ; RK_06 铝壳上料升降气缸下降条件
ANDNOT 514.01  ; RK_06 铝壳上料升降气缸上升条件
LDNOT 814.00  ; RK_06 铝壳上料升降气缸下降位标志[0014.00]
LD 114.01  ; RK_06 铝壳上料升降气缸上升
AND 814.00  ; RK_06 铝壳上料升降气缸下降位标志[0014.00]
ORLD
ANDLD
OUT 414.00  ; RK_06 铝壳上料升降气缸下降[M]
LD TR0
LD 714.01  ; RK_06 铝壳上料升降气缸上升[SW]
LD D1097.05  ; RK_06 铝壳上料升降气缸上升（复位）
ANDNOT D1086.04  ; RK_06 电池上下料机构铝壳上料升降气缸上升1（步）
ANDNOT D1089.04  ; RK_06 电池上下料机构铝壳上料升降气缸上升2（步）
ANDNOT D1086.02  ; RK_06 电池上下料机构铝壳上料升降气缸下降1（步）
ANDNOT D1089.02  ; RK_06 电池上下料机构铝壳上料升降气缸下降2（步）
ORLD
ANDLD
DIFU(013) 314.01  ; RK_06 铝壳上料升降气缸上升[Pls]
LD TR0
LD 314.01  ; RK_06 铝壳上料升降气缸上升[Pls]
OR 414.01  ; RK_06 铝壳上料升降气缸上升[M]
ANDLD
ANDNOT 314.00  ; RK_06 铝壳上料升降气缸下降[Pls]
ANDNOT 514.01  ; RK_06 铝壳上料升降气缸上升条件
ANDNOT 514.00  ; RK_06 铝壳上料升降气缸下降条件
LDNOT 814.01  ; RK_06 铝壳上料升降气缸上升位标志[0014.01]
LD 114.00  ; RK_06 铝壳上料升降气缸下降
AND 814.01  ; RK_06 铝壳上料升降气缸上升位标志[0014.01]
ORLD
ANDLD
OUT 414.01  ; RK_06 铝壳上料升降气缸上升[M]

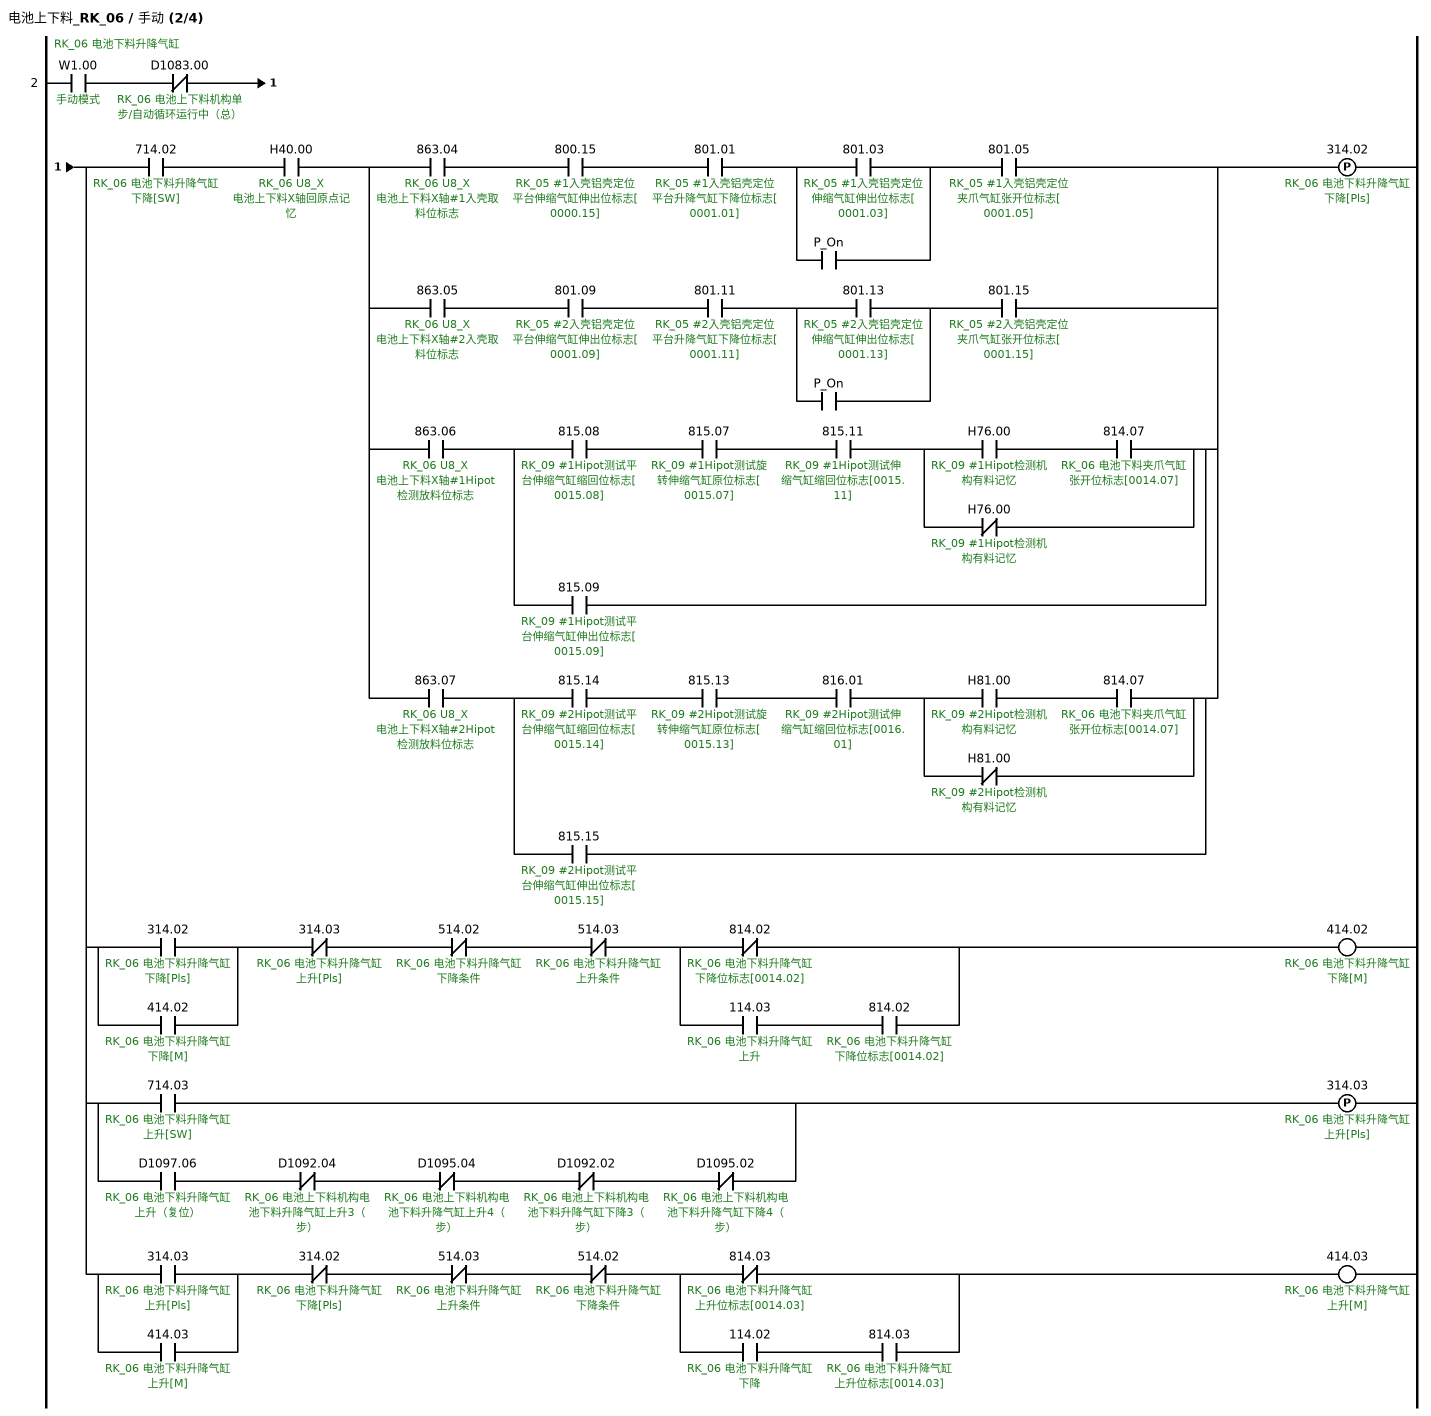
; rung 2: RK_06 电池下料升降气缸
LD W1.00  ; 手动模式
ANDNOT D1083.00  ; RK_06 电池上下料机构单步/自动循环运行中（总）
OUT TR0
AND 714.02  ; RK_06 电池下料升降气缸下降[SW]
AND H40.00  ; RK_06 U8_X 电池上下料X轴回原点记忆
LD 863.04  ; RK_06 U8_X 电池上下料X轴#1入壳取料位标志
AND 800.15  ; RK_05 #1入壳铝壳定位平台伸缩气缸伸出位标志[0000.15]
AND 801.01  ; RK_05 #1入壳铝壳定位平台升降气缸下降位标志[0001.01]
LD 801.03  ; RK_05 #1入壳铝壳定位伸缩气缸伸出位标志[0001.03]
OR P_On
ANDLD
AND 801.05  ; RK_05 #1入壳铝壳定位夹爪气缸张开位标志[0001.05]
LD 863.05  ; RK_06 U8_X 电池上下料X轴#2入壳取料位标志
AND 801.09  ; RK_05 #2入壳铝壳定位平台伸缩气缸伸出位标志[0001.09]
AND 801.11  ; RK_05 #2入壳铝壳定位平台升降气缸下降位标志[0001.11]
LD 801.13  ; RK_05 #2入壳铝壳定位伸缩气缸伸出位标志[0001.13]
OR P_On
ANDLD
AND 801.15  ; RK_05 #2入壳铝壳定位夹爪气缸张开位标志[0001.15]
ORLD
LD 863.06  ; RK_06 U8_X 电池上下料X轴#1Hipot检测放料位标志
LD 815.08  ; RK_09 #1Hipot测试平台伸缩气缸缩回位标志[0015.08]
AND 815.07  ; RK_09 #1Hipot测试旋转伸缩气缸原位标志[0015.07]
AND 815.11  ; RK_09 #1Hipot测试伸缩气缸缩回位标志[0015.11]
LD H76.00  ; RK_09 #1Hipot检测机构有料记忆
AND 814.07  ; RK_06 电池下料夹爪气缸张开位标志[0014.07]
ORNOT H76.00  ; RK_09 #1Hipot检测机构有料记忆
ANDLD
OR 815.09  ; RK_09 #1Hipot测试平台伸缩气缸伸出位标志[0015.09]
ANDLD
ORLD
LD 863.07  ; RK_06 U8_X 电池上下料X轴#2Hipot检测放料位标志
LD 815.14  ; RK_09 #2Hipot测试平台伸缩气缸缩回位标志[0015.14]
AND 815.13  ; RK_09 #2Hipot测试旋转伸缩气缸原位标志[0015.13]
AND 816.01  ; RK_09 #2Hipot测试伸缩气缸缩回位标志[0016.01]
LD H81.00  ; RK_09 #2Hipot检测机构有料记忆
AND 814.07  ; RK_06 电池下料夹爪气缸张开位标志[0014.07]
ORNOT H81.00  ; RK_09 #2Hipot检测机构有料记忆
ANDLD
OR 815.15  ; RK_09 #2Hipot测试平台伸缩气缸伸出位标志[0015.15]
ANDLD
ORLD
ANDLD
DIFU(013) 314.02  ; RK_06 电池下料升降气缸下降[Pls]
LD TR0
LD 314.02  ; RK_06 电池下料升降气缸下降[Pls]
OR 414.02  ; RK_06 电池下料升降气缸下降[M]
ANDLD
ANDNOT 314.03  ; RK_06 电池下料升降气缸上升[Pls]
ANDNOT 514.02  ; RK_06 电池下料升降气缸下降条件
ANDNOT 514.03  ; RK_06 电池下料升降气缸上升条件
LDNOT 814.02  ; RK_06 电池下料升降气缸下降位标志[0014.02]
LD 114.03  ; RK_06 电池下料升降气缸上升
AND 814.02  ; RK_06 电池下料升降气缸下降位标志[0014.02]
ORLD
ANDLD
OUT 414.02  ; RK_06 电池下料升降气缸下降[M]
LD TR0
LD 714.03  ; RK_06 电池下料升降气缸上升[SW]
LD D1097.06  ; RK_06 电池下料升降气缸上升（复位）
ANDNOT D1092.04  ; RK_06 电池上下料机构电池下料升降气缸上升3（步）
ANDNOT D1095.04  ; RK_06 电池上下料机构电池下料升降气缸上升4（步）
ANDNOT D1092.02  ; RK_06 电池上下料机构电池下料升降气缸下降3（步）
ANDNOT D1095.02  ; RK_06 电池上下料机构电池下料升降气缸下降4（步）
ORLD
ANDLD
DIFU(013) 314.03  ; RK_06 电池下料升降气缸上升[Pls]
LD TR0
LD 314.03  ; RK_06 电池下料升降气缸上升[Pls]
OR 414.03  ; RK_06 电池下料升降气缸上升[M]
ANDLD
ANDNOT 314.02  ; RK_06 电池下料升降气缸下降[Pls]
ANDNOT 514.03  ; RK_06 电池下料升降气缸上升条件
ANDNOT 514.02  ; RK_06 电池下料升降气缸下降条件
LDNOT 814.03  ; RK_06 电池下料升降气缸上升位标志[0014.03]
LD 114.02  ; RK_06 电池下料升降气缸下降
AND 814.03  ; RK_06 电池下料升降气缸上升位标志[0014.03]
ORLD
ANDLD
OUT 414.03  ; RK_06 电池下料升降气缸上升[M]

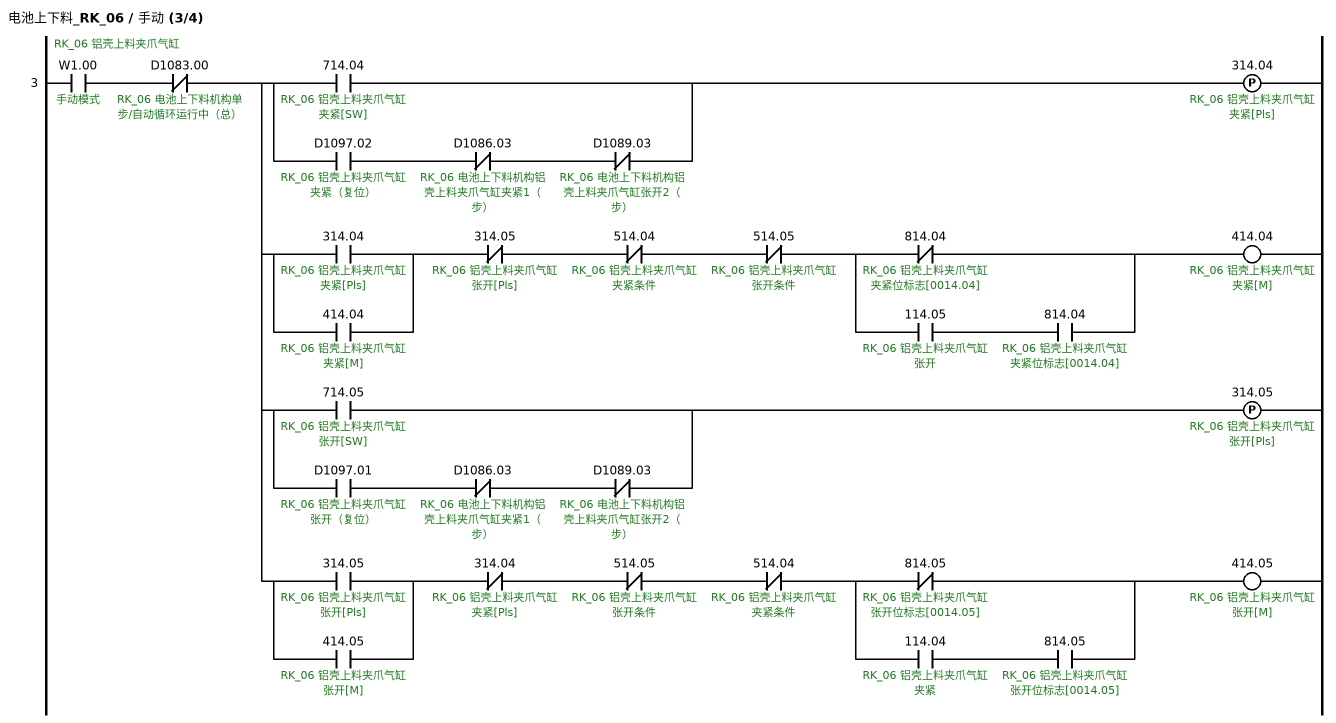
; rung 3: RK_06 铝壳上料夹爪气缸
LD W1.00  ; 手动模式
ANDNOT D1083.00  ; RK_06 电池上下料机构单步/自动循环运行中（总）
OUT TR0
LD 714.04  ; RK_06 铝壳上料夹爪气缸夹紧[SW]
LD D1097.02  ; RK_06 铝壳上料夹爪气缸夹紧（复位）
ANDNOT D1086.03  ; RK_06 电池上下料机构铝壳上料夹爪气缸夹紧1（步）
ANDNOT D1089.03  ; RK_06 电池上下料机构铝壳上料夹爪气缸张开2（步）
ORLD
ANDLD
DIFU(013) 314.04  ; RK_06 铝壳上料夹爪气缸夹紧[Pls]
LD TR0
LD 314.04  ; RK_06 铝壳上料夹爪气缸夹紧[Pls]
OR 414.04  ; RK_06 铝壳上料夹爪气缸夹紧[M]
ANDLD
ANDNOT 314.05  ; RK_06 铝壳上料夹爪气缸张开[Pls]
ANDNOT 514.04  ; RK_06 铝壳上料夹爪气缸夹紧条件
ANDNOT 514.05  ; RK_06 铝壳上料夹爪气缸张开条件
LDNOT 814.04  ; RK_06 铝壳上料夹爪气缸夹紧位标志[0014.04]
LD 114.05  ; RK_06 铝壳上料夹爪气缸张开
AND 814.04  ; RK_06 铝壳上料夹爪气缸夹紧位标志[0014.04]
ORLD
ANDLD
OUT 414.04  ; RK_06 铝壳上料夹爪气缸夹紧[M]
LD TR0
LD 714.05  ; RK_06 铝壳上料夹爪气缸张开[SW]
LD D1097.01  ; RK_06 铝壳上料夹爪气缸张开（复位）
ANDNOT D1086.03  ; RK_06 电池上下料机构铝壳上料夹爪气缸夹紧1（步）
ANDNOT D1089.03  ; RK_06 电池上下料机构铝壳上料夹爪气缸张开2（步）
ORLD
ANDLD
DIFU(013) 314.05  ; RK_06 铝壳上料夹爪气缸张开[Pls]
LD TR0
LD 314.05  ; RK_06 铝壳上料夹爪气缸张开[Pls]
OR 414.05  ; RK_06 铝壳上料夹爪气缸张开[M]
ANDLD
ANDNOT 314.04  ; RK_06 铝壳上料夹爪气缸夹紧[Pls]
ANDNOT 514.05  ; RK_06 铝壳上料夹爪气缸张开条件
ANDNOT 514.04  ; RK_06 铝壳上料夹爪气缸夹紧条件
LDNOT 814.05  ; RK_06 铝壳上料夹爪气缸张开位标志[0014.05]
LD 114.04  ; RK_06 铝壳上料夹爪气缸夹紧
AND 814.05  ; RK_06 铝壳上料夹爪气缸张开位标志[0014.05]
ORLD
ANDLD
OUT 414.05  ; RK_06 铝壳上料夹爪气缸张开[M]

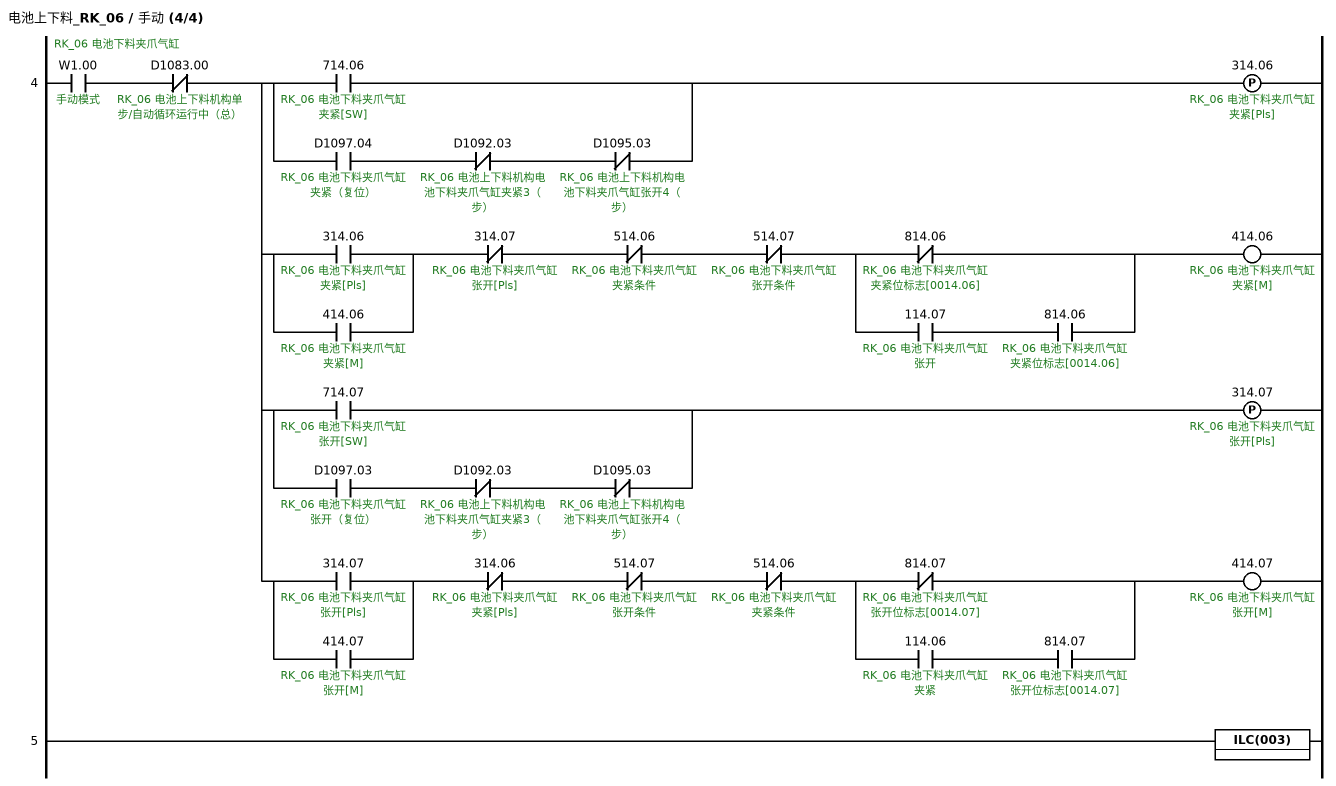
; rung 4: RK_06 电池下料夹爪气缸
LD W1.00  ; 手动模式
ANDNOT D1083.00  ; RK_06 电池上下料机构单步/自动循环运行中（总）
OUT TR0
LD 714.06  ; RK_06 电池下料夹爪气缸夹紧[SW]
LD D1097.04  ; RK_06 电池下料夹爪气缸夹紧（复位）
ANDNOT D1092.03  ; RK_06 电池上下料机构电池下料夹爪气缸夹紧3（步）
ANDNOT D1095.03  ; RK_06 电池上下料机构电池下料夹爪气缸张开4（步）
ORLD
ANDLD
DIFU(013) 314.06  ; RK_06 电池下料夹爪气缸夹紧[Pls]
LD TR0
LD 314.06  ; RK_06 电池下料夹爪气缸夹紧[Pls]
OR 414.06  ; RK_06 电池下料夹爪气缸夹紧[M]
ANDLD
ANDNOT 314.07  ; RK_06 电池下料夹爪气缸张开[Pls]
ANDNOT 514.06  ; RK_06 电池下料夹爪气缸夹紧条件
ANDNOT 514.07  ; RK_06 电池下料夹爪气缸张开条件
LDNOT 814.06  ; RK_06 电池下料夹爪气缸夹紧位标志[0014.06]
LD 114.07  ; RK_06 电池下料夹爪气缸张开
AND 814.06  ; RK_06 电池下料夹爪气缸夹紧位标志[0014.06]
ORLD
ANDLD
OUT 414.06  ; RK_06 电池下料夹爪气缸夹紧[M]
LD TR0
LD 714.07  ; RK_06 电池下料夹爪气缸张开[SW]
LD D1097.03  ; RK_06 电池下料夹爪气缸张开（复位）
ANDNOT D1092.03  ; RK_06 电池上下料机构电池下料夹爪气缸夹紧3（步）
ANDNOT D1095.03  ; RK_06 电池上下料机构电池下料夹爪气缸张开4（步）
ORLD
ANDLD
DIFU(013) 314.07  ; RK_06 电池下料夹爪气缸张开[Pls]
LD TR0
LD 314.07  ; RK_06 电池下料夹爪气缸张开[Pls]
OR 414.07  ; RK_06 电池下料夹爪气缸张开[M]
ANDLD
ANDNOT 314.06  ; RK_06 电池下料夹爪气缸夹紧[Pls]
ANDNOT 514.07  ; RK_06 电池下料夹爪气缸张开条件
ANDNOT 514.06  ; RK_06 电池下料夹爪气缸夹紧条件
LDNOT 814.07  ; RK_06 电池下料夹爪气缸张开位标志[0014.07]
LD 114.06  ; RK_06 电池下料夹爪气缸夹紧
AND 814.07  ; RK_06 电池下料夹爪气缸张开位标志[0014.07]
ORLD
ANDLD
OUT 414.07  ; RK_06 电池下料夹爪气缸张开[M]
; rung 5
ILC(003)

### Section 自动

